
FUNCTION_BLOCK "A_3125_MXZ01MA_Code"
TITLE =A_3125_MXZ01MA FAN 1
//COPYRIGHT:     (C) 2009  BUHLER AG, CH-9240 UZWIL, SWITZERLAND
//
//PRODUCT:       WinCoS_BIW01_09
//
//TITLE:         FAN 1
//
//--------------------------------------------------------------------------------
//
//IDENT:         AUTHOR:             DEPT:                             DATE:
//
//P01_FB1018.1.0 K.Renz              CSB41                             20.Mai.2010
//               1st Release
//
//--------------------------------------------------------------------------------
//
//PURPOSE:
//
//MANUAL :
//
//RESTRICTIONS:
//
//--------------------------------------------------------------------------------
AUTHOR : KR
FAMILY : USW
VERSION : 0.0


VAR
  Ma : "GCS7_M_FB50_Data";	// Machine
  A_3125_KCU04 : "GCS7_E_DigInput";	// Mon1: DigInpCont
  Mon2 : "GCS7_E_DigInput";	// Mon2: DigInpCont
  Mon3 : "GCS7_E_DigInput";	// spare
  A_3125_BSA07 : "GCS7_E_DigInput";	// Mon4: DigInpCont
  Mon5 : "GCS7_E_DigInput";	// spare
  Mon6 : "GCS7_E_DigInput";	// spare
  A_3125_MXZ01 : "GCS7_E_Motor";	// Motor: Motor
END_VAR
BEGIN
NETWORK
TITLE =Call SSW

      UC    "GCS7_M_Motor6Mon";
END_FUNCTION_BLOCK


FUNCTION_BLOCK "A_3126_MXZ01MA_Code"
TITLE =A_3126_MXZ01MA FAN 2
//COPYRIGHT:     (C) 2009  BUHLER AG, CH-9240 UZWIL, SWITZERLAND
//
//PRODUCT:       WinCoS_BIW01_09
//
//TITLE:         FAN 2
//
//--------------------------------------------------------------------------------
//
//IDENT:         AUTHOR:             DEPT:                             DATE:
//
//P01_FB1019.1.0 K.Renz              CSB41                             20.Mai.2010
//               1st Release
//
//--------------------------------------------------------------------------------
//
//PURPOSE:
//
//MANUAL :
//
//RESTRICTIONS:
//
//--------------------------------------------------------------------------------
AUTHOR : KR
FAMILY : USW
VERSION : 0.0


VAR
  Ma : "GCS7_M_FB50_Data";	// Machine
  A_3126_KCU04 : "GCS7_E_DigInput";	// Mon1: DigInpCont
  Mon2 : "GCS7_E_DigInput";	// Mon2: DigInpCont
  Mon3 : "GCS7_E_DigInput";	// spare
  A_3126_BSA07 : "GCS7_E_DigInput";	// Mon4: DigInpCont
  Mon5 : "GCS7_E_DigInput";	// spare
  Mon6 : "GCS7_E_DigInput";	// spare
  A_3126_MXZ01 : "GCS7_E_Motor";	// Motor: Motor
END_VAR
BEGIN
NETWORK
TITLE =Call SSW

      UC    "GCS7_M_Motor6Mon";
END_FUNCTION_BLOCK


FUNCTION_BLOCK "A_3914_MXZ01MA_Code"
TITLE =A_3125_MXZ02MA GETRIEBEÖLPUMPE FAN 1
//COPYRIGHT:     (C) 2009  BUHLER AG, CH-9240 UZWIL, SWITZERLAND
//
//PRODUCT:       WinCoS_BIW01_09
//
//TITLE:         GETRIEBEÖLPUMPE FAN 1
//
//--------------------------------------------------------------------------------
//
//IDENT:         AUTHOR:             DEPT:                             DATE:
//
//P01_FB1025.1.0 K.Renz              CSB41                             20.Mai.2010
//               1st Release
//
//--------------------------------------------------------------------------------
//
//PURPOSE:
//
//MANUAL :
//
//RESTRICTIONS:
//
//--------------------------------------------------------------------------------
AUTHOR : KR
FAMILY : USW
VERSION : 0.0


VAR
  Ma : "GCS7_M_FB50_Data";	// Machine
  A_3125_BFT09 : "GCS7_E_DigInput";	// Mon1: DigInpCont
  Mon2 : "GCS7_E_DigInput";	// Mon2: DigInpCont
  Mon3 : "GCS7_E_DigInput";	// spare
  Mon4 : "GCS7_E_DigInput";	// spare
  Mon5 : "GCS7_E_DigInput";	// spare
  Mon6 : "GCS7_E_DigInput";	// spare
  A_3125_MXZ02 : "GCS7_E_Motor";	// Motor: Motor
END_VAR
BEGIN
NETWORK
TITLE =Call SSW

      UC    "GCS7_M_Motor6Mon";
END_FUNCTION_BLOCK


FUNCTION_BLOCK FB 1065
TITLE =A_3126_MXZ02MA GETRIEBEÖLPUMPE FAN 2
//COPYRIGHT:     (C) 2009  BUHLER AG, CH-9240 UZWIL, SWITZERLAND
//
//PRODUCT:       WinCoS_BIW01_09
//
//TITLE:         GETRIEBEÖLPUMPE FAN 2
//
//--------------------------------------------------------------------------------
//
//IDENT:         AUTHOR:             DEPT:                             DATE:
//
//P01_FB1065.1.0 K.Renz              CSB41                             20.Mai.2010
//               1st Release
//
//--------------------------------------------------------------------------------
//
//PURPOSE:
//
//MANUAL :
//
//RESTRICTIONS:
//
//--------------------------------------------------------------------------------
AUTHOR : KR
FAMILY : USW
VERSION : 0.0


VAR
  Ma : "GCS7_M_FB50_Data";	// Machine
  A_3225_BFT09 : "GCS7_E_DigInput";	// Mon1: DigInpCont
  Mon2 : "GCS7_E_DigInput";	// Mon2: DigInpCont
  Mon3 : "GCS7_E_DigInput";	// spare
  Mon4 : "GCS7_E_DigInput";	// spare
  Mon5 : "GCS7_E_DigInput";	// spare
  Mon6 : "GCS7_E_DigInput";	// spare
  A_3225_MXZ02 : "GCS7_E_Motor";	// Motor: Motor
END_VAR
BEGIN
NETWORK
TITLE =Call SSW

      UC    "GCS7_M_Motor6Mon";
END_FUNCTION_BLOCK


FUNCTION_BLOCK "G271M_Code"
TITLE =G271M FAN KILN 1
//COPYRIGHT:    (C) 2009  BUHLER AG, CH-9240 UZWIL, SWITZERLAND
//
//PRODUCT:      WinCoS_BIW01_09
//
//TITLE:        FAN KILN 1
//                Machine group control
//                Maschinengruppensteuerung
//
//--------------------------------------------------------------------------------
//
//IDENT:        AUTHOR:             DEPT:                              DATE:
//
//P01_FB371.1.0 K.Renz              CSB41                              20.Mai.2010
//             1st Release
//
//--------------------------------------------------------------------------------
//
//PURPOSE:
//
//MANUAL :
//
//RESTRICTIONS:
//
//--------------------------------------------------------------------------------
AUTHOR : KR
FAMILY : USW
VERSION : 9.9


VAR
  Gr : "GCS7_GrpCtrlSub";	//Standard interface to group
  InOutValue1 : DINT ;	//Data for user
  InOutValue2 : DINT ;	//Data for user
  OutWayConflict : BOOL ;	//Data for user
  OutSelectionOk : BOOL ;	//Data for user
  CmdNewValue : BOOL ;	//Data for user
  CmdNewJob : BOOL ;	//Data for user
  OutCodeOK : BOOL ;	//Data for user
  InEndOfJob : BOOL ;	//Data for user
  staWayOk : BOOL ;	//Data for user
  EdgeStartRelease : BOOL ;	//Data for user
  USW8 : BOOL ;	//Data for user
  USW9 : BOOL ;	//Data for user
  USW10 : BOOL ;	//Data for user
  USW11 : BOOL ;	//Data for user
  USW12 : BOOL ;	//Data for user
  USW13 : BOOL ;	//Data for user
  USW14 : BOOL ;	//Data for user
  USW15 : BOOL ;	//Data for user
  A_3125_KCU04AI1 : "GCS7_E_AnalogInput";	// AnaInp
  A_3125_KCU04AI2 : "GCS7_E_AnalogInput";	// AnaInp
  A_3125_BTE05 : "GCS7_E_AnalogInput";	// AnaInp
  A_3125_BTE06 : "GCS7_E_AnalogInput";	// AnaInp
  A_3125_MXZ01MA : "A_3125_MXZ01MA_Code";	// Motor+6DI
  A_3125_TSC01_COM : "SSA_ABB";	// FU_ABB
  A_3125_TSC01_AC : "GCS7_E_AnalogInput";	// AnaInp
  A_3125_TSC01_AF : "GCS7_E_AnalogInput";	// AnaInp
  A_3125_TSC01_AT : "GCS7_E_AnalogInput";	// AnaInp
  A_3125_TSC01_AP : "GCS7_E_AnalogInput";	// AnaInp
  A_3126_KCU04AI1 : "GCS7_E_AnalogInput";	// AnaInp
  A_3126_KCU04AI2 : "GCS7_E_AnalogInput";	// AnaInp
  A_3126_BTE05 : "GCS7_E_AnalogInput";	// AnaInp
  A_3126_BTE06 : "GCS7_E_AnalogInput";	// AnaInp
  A_3126_MXZ01MA : "A_3126_MXZ01MA_Code";	// Motor+6DI
  A_3126_TSC01_COM : "SSA_ABB";	// FU_ABB
  A_3126_TSC01_AC : "GCS7_E_AnalogInput";	// AnaInp
  A_3126_TSC01_AF : "GCS7_E_AnalogInput";	// AnaInp
  A_3126_TSC01_AP : "GCS7_E_AnalogInput";	// AnaInp
  A_3126_TSC01_AT : "GCS7_E_AnalogInput";	// AnaInp
  A_3125_TSC01 : "GCS7_E_DigInput";	// DigInpCont
  A_3126_TSC01 : "GCS7_E_DigInput";	// DigInpCont
  A_3125_MXZ02MA : "A_3914_MXZ01MA_Code";	// Motor+6DI
  A_3126_MXZ02MA : FB 1065;	// Motor+6DI
END_VAR
VAR_TEMP
  tmpEnable : BOOL ;
  tmpFlag : BOOL ;
  tmpCmdNext : BOOL ;
  tmpLocal : BOOL ;
  tmpAspOk : BOOL ;
  tmpHWStop : BOOL ;
  tmpInstanzDBNo : INT ;
END_VAR
BEGIN
NETWORK
TITLE =

NETWORK
TITLE =Read command from group control
//Parameter
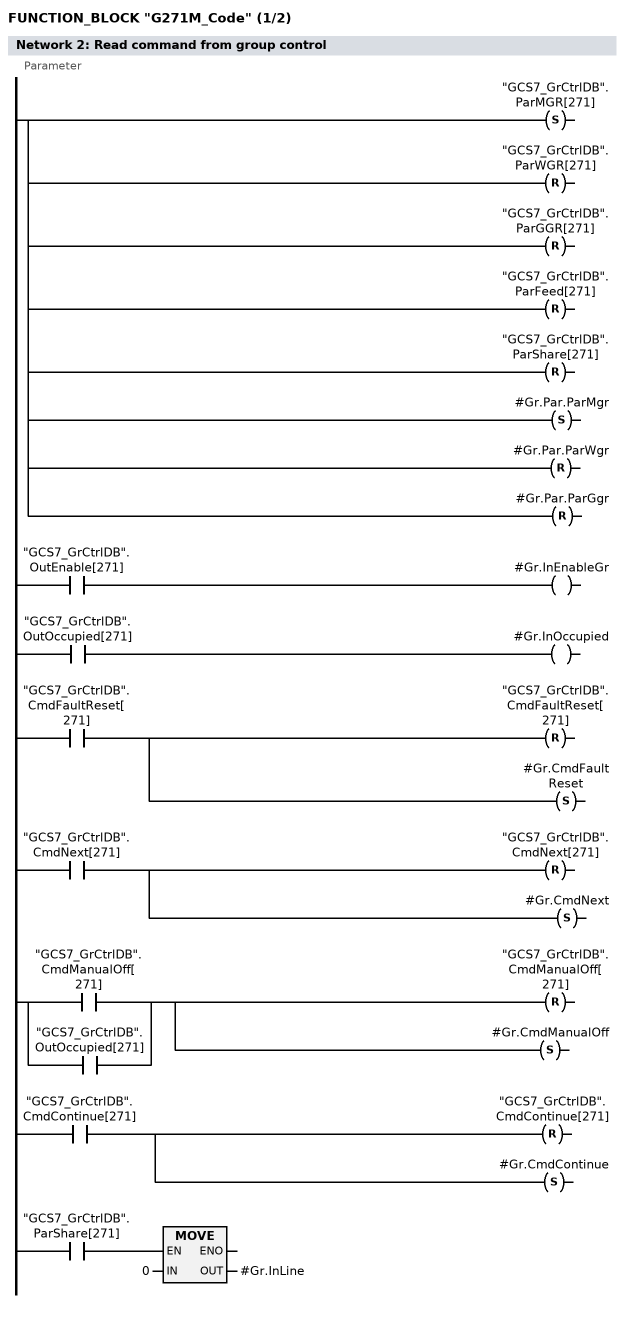
      SET   ;
      S     "GCS7_GrCtrlDB".ParMGR[271];
      R     "GCS7_GrCtrlDB".ParWGR[271];
      R     "GCS7_GrCtrlDB".ParGGR[271];
      R     "GCS7_GrCtrlDB".ParFeed[271];
      R     "GCS7_GrCtrlDB".ParShare[271];
      S     #Gr.Par.ParMgr;
      R     #Gr.Par.ParWgr;
      R     #Gr.Par.ParGgr;
//Command
      U     "GCS7_GrCtrlDB".OutEnable[271];
      =     #Gr.InEnableGr;
      U     "GCS7_GrCtrlDB".OutOccupied[271];
      =     #Gr.InOccupied;
      U     "GCS7_GrCtrlDB".CmdFaultReset[271];
      R     "GCS7_GrCtrlDB".CmdFaultReset[271];
      S     #Gr.CmdFaultReset;
      U     "GCS7_GrCtrlDB".CmdNext[271];
      R     "GCS7_GrCtrlDB".CmdNext[271];
      S     #Gr.CmdNext;
      U     "GCS7_GrCtrlDB".CmdManualOff[271];
      O     "GCS7_GrCtrlDB".OutOccupied[271];
      R     "GCS7_GrCtrlDB".CmdManualOff[271];
      S     #Gr.CmdManualOff;
      U     "GCS7_GrCtrlDB".CmdContinue[271];
      R     "GCS7_GrCtrlDB".CmdContinue[271];
      S     #Gr.CmdContinue;
//Init Line Number
      U     "GCS7_GrCtrlDB".ParShare[271];
      SPBN  WE00;
      L     0;
      T     #Gr.InLine;
WE00: NOP   0;
NETWORK
TITLE =Call Methode Control
// 1. Handle Interface PCControl
// 2. Prepare mode --> ModePassive,ModeActive,ModeIdling
// 3. Reset global flags of the group
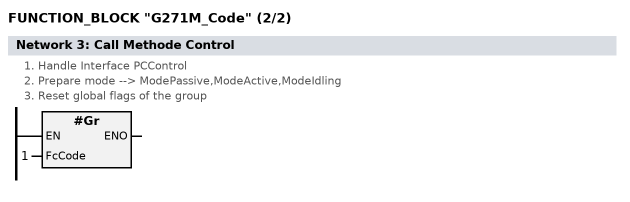
      CALL #Gr (
           FcCode                   := 1);
NETWORK
TITLE =Restart Idling Time

      L     #Gr.Par.ParIdling;
      L     2;
      >=I   ;
      SPB   IdTm;
      T     #Gr.Par.ParIdling;
IdTm: NOP   0;
      CLR   ;
      S     #Gr.CmdRestartIdling;
NETWORK
TITLE =Prepare global flags

NETWORK
TITLE =Set Pattern (Target position)

NETWORK
TITLE =Interlocking WayOk

NETWORK
TITLE =Interlocking Autostart

      CLR   ;
      R     #Gr.OutAutostart;
NETWORK
TITLE =Interlocking Enable
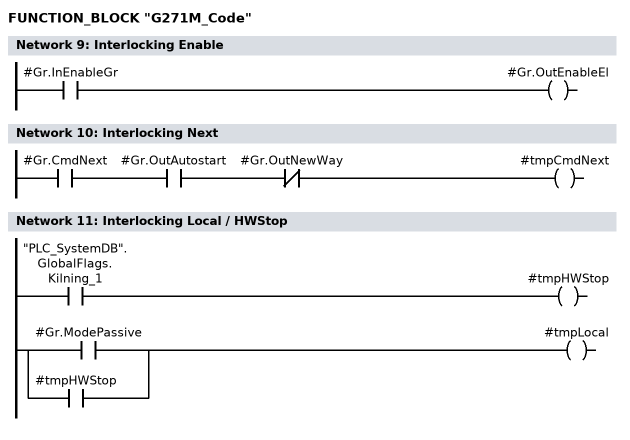

      U     #Gr.InEnableGr;
      =     #Gr.OutEnableEl;

NETWORK
TITLE =Interlocking Next

      U     #Gr.CmdNext;
      U     #Gr.OutAutostart;
      UN    #Gr.OutNewWay;
      =     #tmpCmdNext;

NETWORK
TITLE =Interlocking Local / HWStop

      U     "PLC_SystemDB".GlobalFlags.Kilning_1;
      =     #tmpHWStop;

      U     #Gr.ModePassive;
      O     #tmpHWStop;
      =     #tmpLocal;

NETWORK
TITLE =Interlocking Start Warning

      NOP   0;
//- Restart after fault --
      U     #Gr.CmdFaultReset;
      U     #Gr.VarFault;
      S     "SYS_StartWarningDB".Area[10].CmdResetStartWarning;
//- Run Timer --
      AUF   "G271M";
      CALL "GCS7_StartWarning" , "SYS_StartWarningDB" (
           InModeHigher             := FALSE,
           InArea                   := 10,
           InEnable                 := #Gr.OutEnableEl,
           InLocal                  := #tmpLocal,
           InStarted                := #Gr.VarStarted,
           InCmdNext                := #tmpCmdNext,
           OutCmdNext               := #tmpCmdNext,
           OutStartwarning          := #Gr.VarStartwarning);
//- Store Startwarning done  --
//- Reset Autostart --
      U     "SYS_StartWarningDB".TmpArea.OutStartReleaseRunningL;
      FN    #EdgeStartRelease;
      U     #Gr.VarFault;
      R     #Gr.OutAutostart;
NETWORK
TITLE ==A-3125-KCU04AI1 : VIBRATION MONITOR FAN 1 CHANNEL 1

      NOP   0;
//-InLocal---
      U     #tmpLocal;
      =     #A_3125_KCU04AI1.InLocal;
//
//-Monitoring---
      CLR   ;
      =     #A_3125_KCU04AI1.InMonLL;
      CLR   ;
      =     #A_3125_KCU04AI1.InMonL;
      CLR   ;
      =     #A_3125_KCU04AI1.InMonMid;
      CLR   ;
      =     #A_3125_KCU04AI1.InMonH;
      SET   ;
      =     #A_3125_KCU04AI1.InMonHH;
//
//-Read inputs---
      L     "A_3125_KCU04_AI1";
      T     #A_3125_KCU04AI1.InpValue;
      U     "PLC_SystemDB".GlobalFlags.Kilning_1;
      =     #A_3125_KCU04AI1.InHWStop;
      U     "PLC_DPInfo".Master[1].SlavesError[92];
      =     #A_3125_KCU04AI1.InDPFault;
//
//-Set Parameters---
//
//-Call object control---
      CALL #A_3125_KCU04AI1 ;
//
//-Write outputs---
NETWORK
TITLE ==A-3125-KCU04AI2 : VIBRATION MONITOR FAN 1 CHANNEL 2

      NOP   0;
//-InLocal---
      U     #tmpLocal;
      =     #A_3125_KCU04AI2.InLocal;
//
//-Monitoring---
      CLR   ;
      =     #A_3125_KCU04AI2.InMonLL;
      CLR   ;
      =     #A_3125_KCU04AI2.InMonL;
      CLR   ;
      =     #A_3125_KCU04AI2.InMonMid;
      CLR   ;
      =     #A_3125_KCU04AI2.InMonH;
      SET   ;
      =     #A_3125_KCU04AI2.InMonHH;
//
//-Read inputs---
      L     "A_3125_KCU04_AI2";
      T     #A_3125_KCU04AI2.InpValue;
      U     "PLC_SystemDB".GlobalFlags.Kilning_1;
      =     #A_3125_KCU04AI2.InHWStop;
      U     "PLC_DPInfo".Master[1].SlavesError[92];
      =     #A_3125_KCU04AI2.InDPFault;
//
//-Set Parameters---
//
//-Call object control---
      CALL #A_3125_KCU04AI2 ;
//
//-Write outputs---
NETWORK
TITLE ==A-3125-BTE05 : TEMPERATURE BEARING TEMPERATUR SENSOR

      NOP   0;
//-InLocal---
      U     #tmpLocal;
      =     #A_3125_BTE05.InLocal;
//
//-Monitoring---
      CLR   ;
      =     #A_3125_BTE05.InMonLL;
      CLR   ;
      =     #A_3125_BTE05.InMonL;
      CLR   ;
      =     #A_3125_BTE05.InMonMid;
      CLR   ;
      =     #A_3125_BTE05.InMonH;
      SET   ;
      =     #A_3125_BTE05.InMonHH;
//
//-Read inputs---
      L     "A_3125_BTE05_AI1";
      T     #A_3125_BTE05.InpValue;
      U     "PLC_SystemDB".GlobalFlags.Kilning_1;
      =     #A_3125_BTE05.InHWStop;
      U     "PLC_DPInfo".Master[1].SlavesError[92];
      =     #A_3125_BTE05.InDPFault;
//
//-Set Parameters---
//
//-Call object control---
      CALL #A_3125_BTE05 ;
//
//-Write outputs---
NETWORK
TITLE ==A-3125-BTE06 : TEMPERATURE BEARING TEMPERATUR SENSOR

      NOP   0;
//-InLocal---
      U     #tmpLocal;
      =     #A_3125_BTE06.InLocal;
//
//-Monitoring---
      CLR   ;
      =     #A_3125_BTE06.InMonLL;
      CLR   ;
      =     #A_3125_BTE06.InMonL;
      CLR   ;
      =     #A_3125_BTE06.InMonMid;
      CLR   ;
      =     #A_3125_BTE06.InMonH;
      SET   ;
      =     #A_3125_BTE06.InMonHH;
//
//-Read inputs---
      L     "A_3125_BTE06_AI1";
      T     #A_3125_BTE06.InpValue;
      U     "PLC_SystemDB".GlobalFlags.Kilning_1;
      =     #A_3125_BTE06.InHWStop;
      U     "PLC_DPInfo".Master[1].SlavesError[92];
      =     #A_3125_BTE06.InDPFault;
//
//-Set Parameters---
//
//-Call object control---
      CALL #A_3125_BTE06 ;
//
//-Write outputs---
NETWORK
TITLE ==A-3125-MXZ02MA : GETRIEBEÖLPUMPE FAN 1
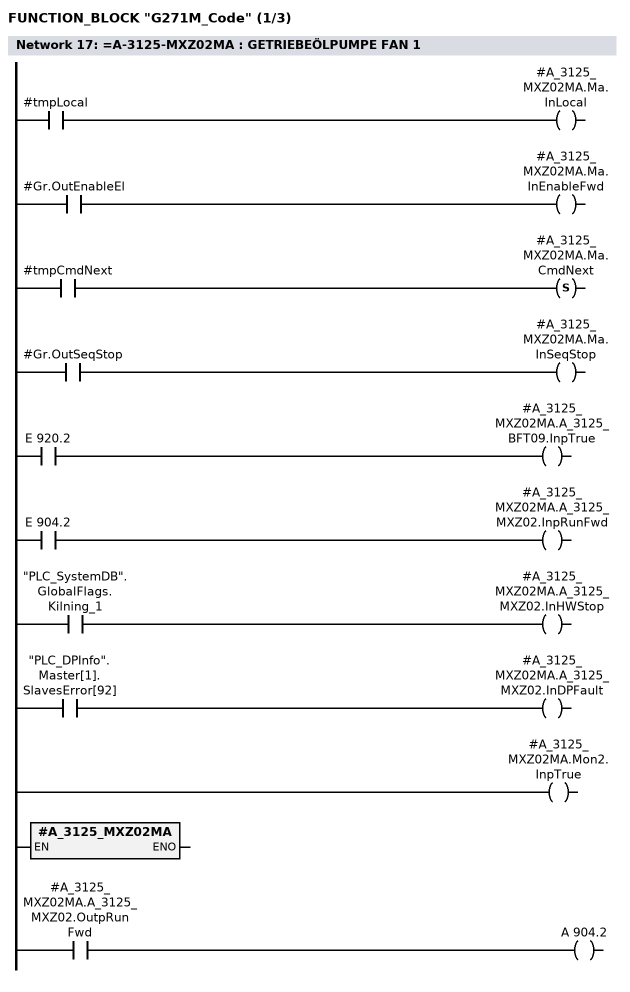

      NOP   0;
//-InLocal---
      U     #tmpLocal;
      =     #A_3125_MXZ02MA.Ma.InLocal;
//
//-Interlocking---

      U     #Gr.OutEnableEl;
      =     #A_3125_MXZ02MA.Ma.InEnableFwd;
//
      U     #tmpCmdNext;
      S     #A_3125_MXZ02MA.Ma.CmdNext;
//
      U     #Gr.OutSeqStop;
      =     #A_3125_MXZ02MA.Ma.InSeqStop;
//
//=Values and commands of elements===
//-=A-3125-BFT09---
//      CLR
//      S     #A_3125_MXZ02MA.A_3125_BFT09.CmdRunTimeOutTime
//
//-Read inputs of elements---
      U     E    920.2;
      =     #A_3125_MXZ02MA.A_3125_BFT09.InpTrue;
      U     E    904.2;
      =     #A_3125_MXZ02MA.A_3125_MXZ02.InpRunFwd;
      U     "PLC_SystemDB".GlobalFlags.Kilning_1;
      =     #A_3125_MXZ02MA.A_3125_MXZ02.InHWStop;
      U     "PLC_DPInfo".Master[1].SlavesError[92];
      =     #A_3125_MXZ02MA.A_3125_MXZ02.InDPFault;
      SET   ;
      =     #A_3125_MXZ02MA.Mon2.InpTrue;
//
//-Set Parameters---
//
//-Call object control---
      CALL #A_3125_MXZ02MA ;
//
//-Write outputs---
      U     #A_3125_MXZ02MA.A_3125_MXZ02.OutpRunFwd;
      =     A    904.2;
NETWORK
TITLE ==A-3125-MXZ01MA : FAN 1
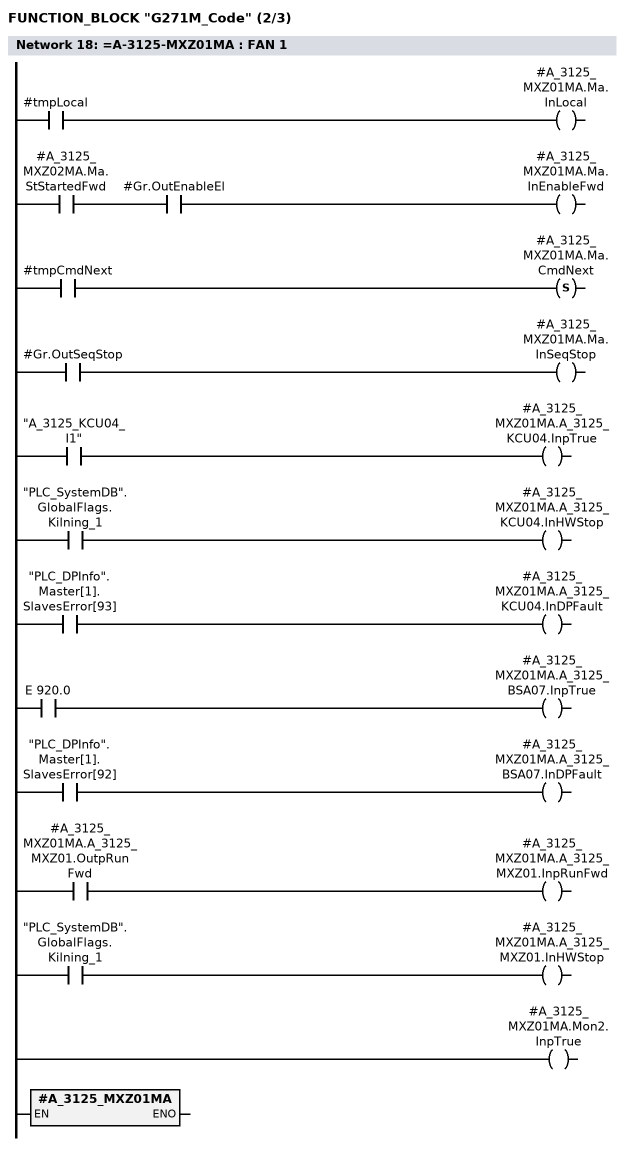

      NOP   0;
//-InLocal---
      U     #tmpLocal;
      =     #A_3125_MXZ01MA.Ma.InLocal;
//
//-Interlocking---
      U     #A_3125_MXZ02MA.Ma.StStartedFwd;
      U     #Gr.OutEnableEl;
      =     #A_3125_MXZ01MA.Ma.InEnableFwd;
//
      U     #tmpCmdNext;
      S     #A_3125_MXZ01MA.Ma.CmdNext;
//
      U     #Gr.OutSeqStop;
      =     #A_3125_MXZ01MA.Ma.InSeqStop;
//
//=Values and commands of elements===
//-=A-3125-KCU04---
//      CLR
//      S     #A_3125_MXZ01MA.A_3125_KCU04.CmdRunTimeOutTime
//-=A-3125-BSA07---
//      CLR
//      S     #A_3125_MXZ01MA.A_3125_BSA07.CmdRunTimeOutTime
//
//-Read inputs of elements---
      U     "A_3125_KCU04_I1";
      =     #A_3125_MXZ01MA.A_3125_KCU04.InpTrue;
      U     "PLC_SystemDB".GlobalFlags.Kilning_1;
      =     #A_3125_MXZ01MA.A_3125_KCU04.InHWStop;
      U     "PLC_DPInfo".Master[1].SlavesError[93];
      =     #A_3125_MXZ01MA.A_3125_KCU04.InDPFault;
      U     E    920.0;
      =     #A_3125_MXZ01MA.A_3125_BSA07.InpTrue;
      U     "PLC_DPInfo".Master[1].SlavesError[92];
      =     #A_3125_MXZ01MA.A_3125_BSA07.InDPFault;
      U     #A_3125_MXZ01MA.A_3125_MXZ01.OutpRunFwd;
      =     #A_3125_MXZ01MA.A_3125_MXZ01.InpRunFwd;
      U     "PLC_SystemDB".GlobalFlags.Kilning_1;
      =     #A_3125_MXZ01MA.A_3125_MXZ01.InHWStop;
      SET   ;
      =     #A_3125_MXZ01MA.Mon2.InpTrue;
//
//-Set Parameters---
//
//-Call object control---
      CALL #A_3125_MXZ01MA ;
//
//-Write outputs---
NETWORK
TITLE ==A-3125-TSC01_COM : FAN 1 FU KOMMUNIKATION
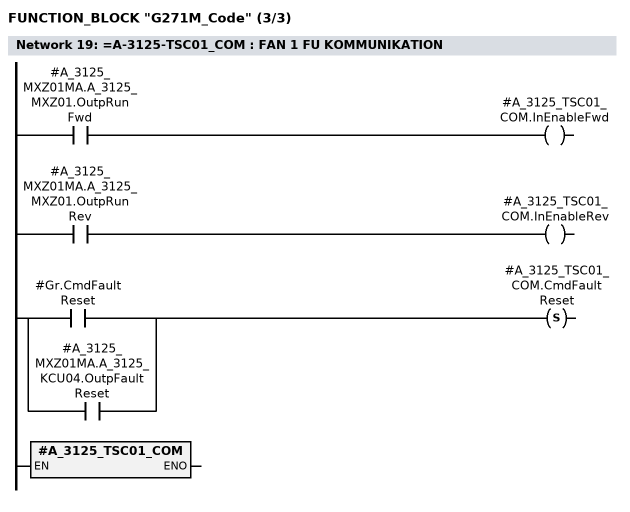

      NOP   0;
      U     #A_3125_MXZ01MA.A_3125_MXZ01.OutpRunFwd;
      =     #A_3125_TSC01_COM.InEnableFwd;
      U     #A_3125_MXZ01MA.A_3125_MXZ01.OutpRunRev;
      =     #A_3125_TSC01_COM.InEnableRev;
      U     #Gr.CmdFaultReset;
      O     #A_3125_MXZ01MA.A_3125_KCU04.OutpFaultReset;
      S     #A_3125_TSC01_COM.CmdFaultReset;
//
//
//-Read inputs---
//
//-Set Parameters---
//
//-Call object control---
      CALL #A_3125_TSC01_COM ;
//
//-Write outputs---
NETWORK
TITLE ==A-3125-TSC01_AC : ACT. CURRENT FAN 1 FU

      NOP   0;
//-InLocal---
      U     #tmpLocal;
      =     #A_3125_TSC01_AC.InLocal;
//
//-Monitoring---
      SET   ;
      =     #A_3125_TSC01_AC.InMonLL;
      CLR   ;
      =     #A_3125_TSC01_AC.InMonL;
      CLR   ;
      =     #A_3125_TSC01_AC.InMonMid;
      CLR   ;
      =     #A_3125_TSC01_AC.InMonH;
      CLR   ;
      =     #A_3125_TSC01_AC.InMonHH;
//
//-Read inputs---
      L     #A_3125_TSC01_COM.Output.SetpointValue01;
      ITD   ;
      DTR   ;
      ABS   ;
      RND   ;
      T     #A_3125_TSC01_AC.InpValue;
      U     "PLC_SystemDB".GlobalFlags.Kilning_1;
      =     #A_3125_TSC01_AC.InHWStop;
//
//-Set Parameters---
//
//-Call object control---
      CALL #A_3125_TSC01_AC ;
//
//-Write outputs---
NETWORK
TITLE ==A-3125-TSC01_AF : ACT. FREQUENCY FAN 1 FU

      NOP   0;
//-InLocal---
      U     #tmpLocal;
      =     #A_3125_TSC01_AF.InLocal;
//
//-Monitoring---
      SET   ;
      =     #A_3125_TSC01_AF.InMonLL;
      CLR   ;
      =     #A_3125_TSC01_AF.InMonL;
      CLR   ;
      =     #A_3125_TSC01_AF.InMonMid;
      CLR   ;
      =     #A_3125_TSC01_AF.InMonH;
      CLR   ;
      =     #A_3125_TSC01_AF.InMonHH;
//
//-Read inputs---
      L     #A_3125_TSC01_COM.Output.SetpointValue01;
      ITD   ;
      DTR   ;
      ABS   ;
      RND   ;
      T     #A_3125_TSC01_AF.InpValue;
      U     "PLC_SystemDB".GlobalFlags.Kilning_1;
      =     #A_3125_TSC01_AF.InHWStop;
//
//-Set Parameters---
//
//-Call object control---
      CALL #A_3125_TSC01_AF ;
//
//-Write outputs---
NETWORK
TITLE ==A-3125-TSC01_AT : ACT. TORQUE FAN 1 FU

      NOP   0;
//-InLocal---
      U     #tmpLocal;
      =     #A_3125_TSC01_AT.InLocal;
//
//-Monitoring---
      CLR   ;
      =     #A_3125_TSC01_AT.InMonLL;
      CLR   ;
      =     #A_3125_TSC01_AT.InMonL;
      CLR   ;
      =     #A_3125_TSC01_AT.InMonMid;
      CLR   ;
      =     #A_3125_TSC01_AT.InMonH;
      CLR   ;
      =     #A_3125_TSC01_AT.InMonHH;
//
//-Read inputs---
      L     #A_3125_TSC01_COM.Output.SetpointValue01;
      ITD   ;
      DTR   ;
      ABS   ;
      RND   ;
      T     #A_3125_TSC01_AT.InpValue;
      U     "PLC_SystemDB".GlobalFlags.Kilning_1;
      =     #A_3125_TSC01_AT.InHWStop;
//
//-Set Parameters---
//
//-Call object control---
      CALL #A_3125_TSC01_AT ;
//
//-Write outputs---
NETWORK
TITLE ==A-3125-TSC01_AP : ACT. POWER FAN 1 FU

      NOP   0;
//-InLocal---
      U     #tmpLocal;
      =     #A_3125_TSC01_AP.InLocal;
//
//-Monitoring---
      CLR   ;
      =     #A_3125_TSC01_AP.InMonLL;
      CLR   ;
      =     #A_3125_TSC01_AP.InMonL;
      CLR   ;
      =     #A_3125_TSC01_AP.InMonMid;
      CLR   ;
      =     #A_3125_TSC01_AP.InMonH;
      CLR   ;
      =     #A_3125_TSC01_AP.InMonHH;
//
//-Read inputs---
      L     #A_3125_TSC01_COM.Output.SetpointValue01;
      ITD   ;
      DTR   ;
      ABS   ;
      RND   ;
      T     #A_3125_TSC01_AP.InpValue;
      U     "PLC_SystemDB".GlobalFlags.Kilning_1;
      =     #A_3125_TSC01_AP.InHWStop;
//
//-Set Parameters---
//
//-Call object control---
      CALL #A_3125_TSC01_AP ;
//
//-Write outputs---
NETWORK
TITLE ==A-3126-KCU04AI1 : VIBRATION MONITOR FAN 2 CHANNEL 1

      NOP   0;
//-InLocal---
      U     #tmpLocal;
      =     #A_3126_KCU04AI1.InLocal;
//
//-Monitoring---
      CLR   ;
      =     #A_3126_KCU04AI1.InMonLL;
      CLR   ;
      =     #A_3126_KCU04AI1.InMonL;
      CLR   ;
      =     #A_3126_KCU04AI1.InMonMid;
      CLR   ;
      =     #A_3126_KCU04AI1.InMonH;
      SET   ;
      =     #A_3126_KCU04AI1.InMonHH;
//
//-Read inputs---
      L     "A_3126_KCU04_AI1";
      T     #A_3126_KCU04AI1.InpValue;
      U     "PLC_SystemDB".GlobalFlags.Kilning_1;
      =     #A_3126_KCU04AI1.InHWStop;
      U     "PLC_DPInfo".Master[1].SlavesError[92];
      =     #A_3126_KCU04AI1.InDPFault;
//
//-Set Parameters---
//
//-Call object control---
      CALL #A_3126_KCU04AI1 ;
//
//-Write outputs---
NETWORK
TITLE ==A-3126-KCU04AI2 : VIBRATION MONITOR FAN 2 CHANNEL 2

      NOP   0;
//-InLocal---
      U     #tmpLocal;
      =     #A_3126_KCU04AI2.InLocal;
//
//-Monitoring---
      CLR   ;
      =     #A_3126_KCU04AI2.InMonLL;
      CLR   ;
      =     #A_3126_KCU04AI2.InMonL;
      CLR   ;
      =     #A_3126_KCU04AI2.InMonMid;
      CLR   ;
      =     #A_3126_KCU04AI2.InMonH;
      SET   ;
      =     #A_3126_KCU04AI2.InMonHH;
//
//-Read inputs---
      L     "A_3126_KCU04_AI2";
      T     #A_3126_KCU04AI2.InpValue;
      U     "PLC_SystemDB".GlobalFlags.Kilning_1;
      =     #A_3126_KCU04AI2.InHWStop;
      U     "PLC_DPInfo".Master[1].SlavesError[92];
      =     #A_3126_KCU04AI2.InDPFault;
//
//-Set Parameters---
//
//-Call object control---
      CALL #A_3126_KCU04AI2 ;
//
//-Write outputs---
NETWORK
TITLE ==A-3126-BTE05 : TEMPERATURE BEARING TEMPERATUR SENSOR

      NOP   0;
//-InLocal---
      U     #tmpLocal;
      =     #A_3126_BTE05.InLocal;
//
//-Monitoring---
      CLR   ;
      =     #A_3126_BTE05.InMonLL;
      CLR   ;
      =     #A_3126_BTE05.InMonL;
      CLR   ;
      =     #A_3126_BTE05.InMonMid;
      CLR   ;
      =     #A_3126_BTE05.InMonH;
      SET   ;
      =     #A_3126_BTE05.InMonHH;
//
//-Read inputs---
      L     "A_3126_BTE05_AI1";
      T     #A_3126_BTE05.InpValue;
      U     "PLC_SystemDB".GlobalFlags.Kilning_1;
      =     #A_3126_BTE05.InHWStop;
      U     "PLC_DPInfo".Master[1].SlavesError[92];
      =     #A_3126_BTE05.InDPFault;
//
//-Set Parameters---
//
//-Call object control---
      CALL #A_3126_BTE05 ;
//
//-Write outputs---
NETWORK
TITLE ==A-3126-BTE06 : TEMPERATURE BEARING TEMPERATUR SENSOR

      NOP   0;
//-InLocal---
      U     #tmpLocal;
      =     #A_3126_BTE06.InLocal;
//
//-Monitoring---
      CLR   ;
      =     #A_3126_BTE06.InMonLL;
      CLR   ;
      =     #A_3126_BTE06.InMonL;
      CLR   ;
      =     #A_3126_BTE06.InMonMid;
      CLR   ;
      =     #A_3126_BTE06.InMonH;
      SET   ;
      =     #A_3126_BTE06.InMonHH;
//
//-Read inputs---
      L     "A_3126_BTE06_AI1";
      T     #A_3126_BTE06.InpValue;
      U     "PLC_SystemDB".GlobalFlags.Kilning_1;
      =     #A_3126_BTE06.InHWStop;
      U     "PLC_DPInfo".Master[1].SlavesError[92];
      =     #A_3126_BTE06.InDPFault;
//
//-Set Parameters---
//
//-Call object control---
      CALL #A_3126_BTE06 ;
//
//-Write outputs---
NETWORK
TITLE ==A-3126-MXZ02MA : GETRIEBEÖLPUMPE FAN 2
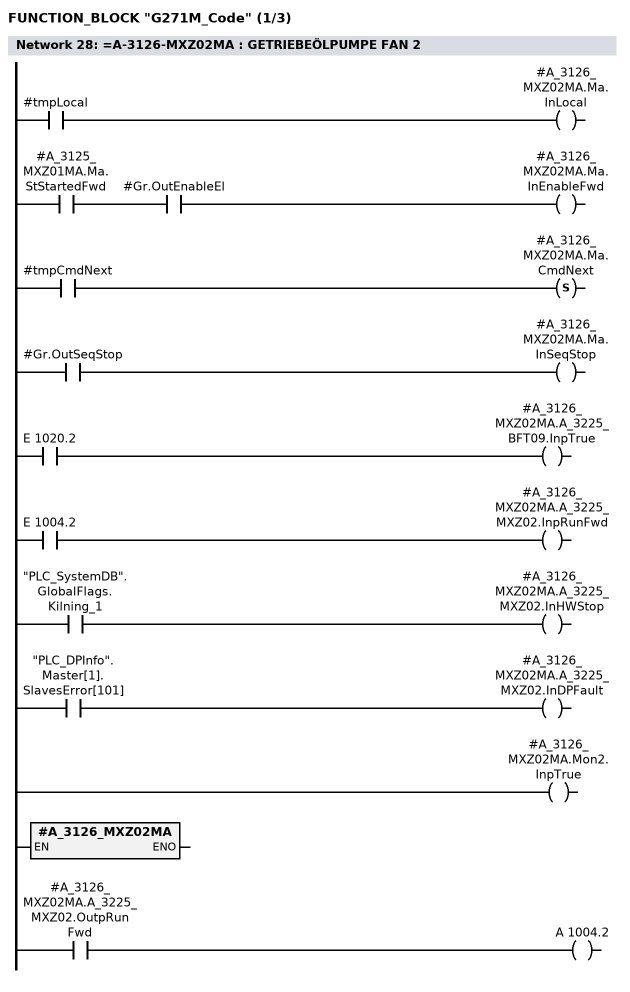

      NOP   0;
//-InLocal---
      U     #tmpLocal;
      =     #A_3126_MXZ02MA.Ma.InLocal;
//
//-Interlocking---
      U     #A_3125_MXZ01MA.Ma.StStartedFwd;
      U     #Gr.OutEnableEl;
      =     #A_3126_MXZ02MA.Ma.InEnableFwd;
//
      U     #tmpCmdNext;
      S     #A_3126_MXZ02MA.Ma.CmdNext;
//
      U     #Gr.OutSeqStop;
      =     #A_3126_MXZ02MA.Ma.InSeqStop;
//
//=Values and commands of elements===
//-=A-3225-BFT09---
//      CLR
//      S     #A_3126_MXZ02MA.A_3225_BFT09.CmdRunTimeOutTime
//
//-Read inputs of elements---
      U     E   1020.2;
      =     #A_3126_MXZ02MA.A_3225_BFT09.InpTrue;
      U     E   1004.2;
      =     #A_3126_MXZ02MA.A_3225_MXZ02.InpRunFwd;
      U     "PLC_SystemDB".GlobalFlags.Kilning_1;
      =     #A_3126_MXZ02MA.A_3225_MXZ02.InHWStop;
      U     "PLC_DPInfo".Master[1].SlavesError[101];
      =     #A_3126_MXZ02MA.A_3225_MXZ02.InDPFault;
      SET   ;
      =     #A_3126_MXZ02MA.Mon2.InpTrue;
//
//-Set Parameters---
//
//-Call object control---
      CALL #A_3126_MXZ02MA ;
//
//-Write outputs---
      U     #A_3126_MXZ02MA.A_3225_MXZ02.OutpRunFwd;
      =     A   1004.2;
NETWORK
TITLE ==A-3126-MXZ01MA : FAN 2
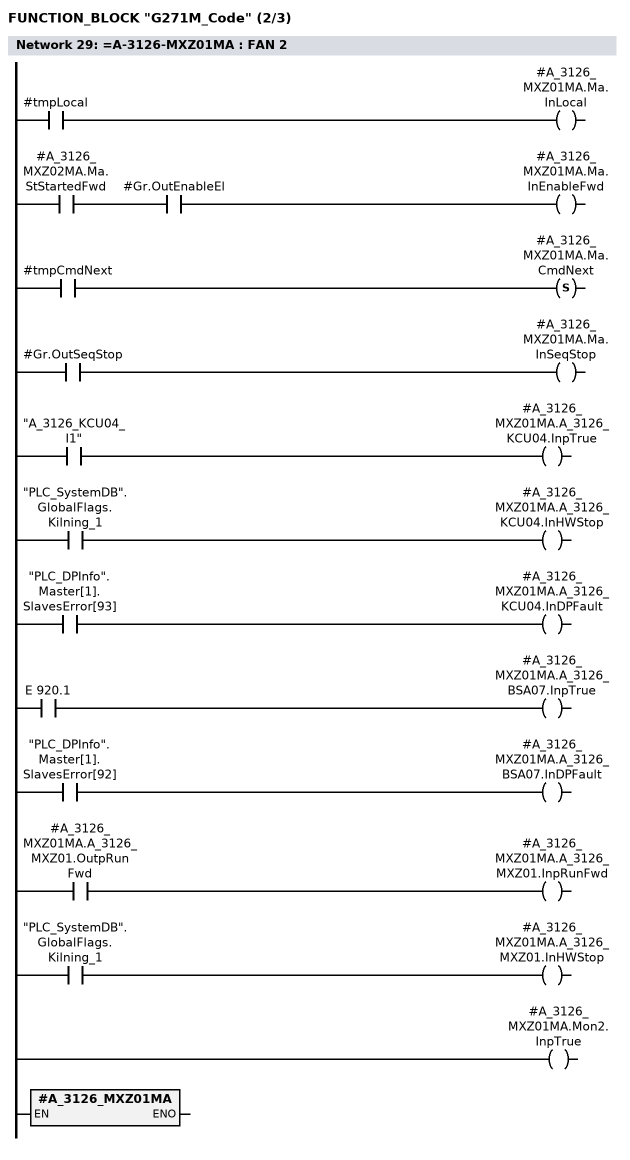

      NOP   0;
//-InLocal---
      U     #tmpLocal;
      =     #A_3126_MXZ01MA.Ma.InLocal;
//
//-Interlocking---
      U     #A_3126_MXZ02MA.Ma.StStartedFwd;
      U     #Gr.OutEnableEl;
      =     #A_3126_MXZ01MA.Ma.InEnableFwd;
//
      U     #tmpCmdNext;
      S     #A_3126_MXZ01MA.Ma.CmdNext;
//
      U     #Gr.OutSeqStop;
      =     #A_3126_MXZ01MA.Ma.InSeqStop;
//
//=Values and commands of elements===
//-=A-3126-KCU04---
//      CLR
//      S     #A_3126_MXZ01MA.A_3126_KCU04.CmdRunTimeOutTime
//-=A-3126-BSA07---
//      CLR
//      S     #A_3126_MXZ01MA.A_3126_BSA07.CmdRunTimeOutTime
//
//-Read inputs of elements---
      U     "A_3126_KCU04_I1";
      =     #A_3126_MXZ01MA.A_3126_KCU04.InpTrue;
      U     "PLC_SystemDB".GlobalFlags.Kilning_1;
      =     #A_3126_MXZ01MA.A_3126_KCU04.InHWStop;
      U     "PLC_DPInfo".Master[1].SlavesError[93];
      =     #A_3126_MXZ01MA.A_3126_KCU04.InDPFault;
      U     E    920.1;
      =     #A_3126_MXZ01MA.A_3126_BSA07.InpTrue;
      U     "PLC_DPInfo".Master[1].SlavesError[92];
      =     #A_3126_MXZ01MA.A_3126_BSA07.InDPFault;
      U     #A_3126_MXZ01MA.A_3126_MXZ01.OutpRunFwd;
      =     #A_3126_MXZ01MA.A_3126_MXZ01.InpRunFwd;
      U     "PLC_SystemDB".GlobalFlags.Kilning_1;
      =     #A_3126_MXZ01MA.A_3126_MXZ01.InHWStop;
      SET   ;
      =     #A_3126_MXZ01MA.Mon2.InpTrue;
//
//-Set Parameters---
//
//-Call object control---
      CALL #A_3126_MXZ01MA ;
//
//-Write outputs---
NETWORK
TITLE ==A-3126-TSC01_COM : FAN 2 FU KOMMUNIKATION
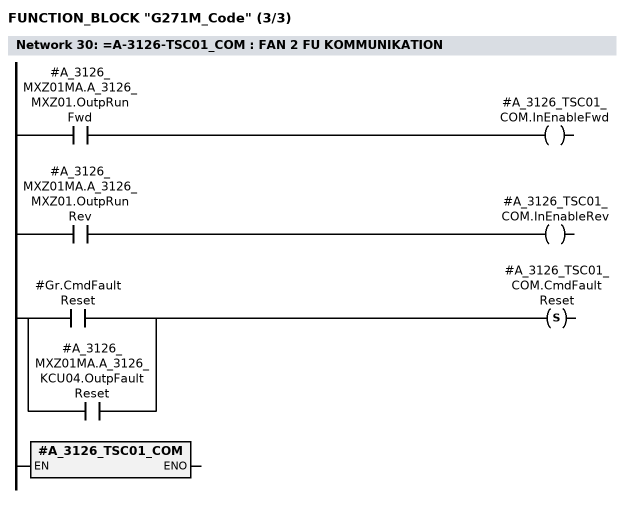

      NOP   0;
      U     #A_3126_MXZ01MA.A_3126_MXZ01.OutpRunFwd;
      =     #A_3126_TSC01_COM.InEnableFwd;
      U     #A_3126_MXZ01MA.A_3126_MXZ01.OutpRunRev;
      =     #A_3126_TSC01_COM.InEnableRev;
      U     #Gr.CmdFaultReset;
      O     #A_3126_MXZ01MA.A_3126_KCU04.OutpFaultReset;
      S     #A_3126_TSC01_COM.CmdFaultReset;
//
//
//-Read inputs---
//
//-Set Parameters---
//
//-Call object control---
      CALL #A_3126_TSC01_COM ;
//
//-Write outputs---
NETWORK
TITLE ==A-3126-TSC01_AC : ACT. CURRENT FAN 2 FU

      NOP   0;
//-InLocal---
      U     #tmpLocal;
      =     #A_3126_TSC01_AC.InLocal;
//
//-Monitoring---
      SET   ;
      =     #A_3126_TSC01_AC.InMonLL;
      CLR   ;
      =     #A_3126_TSC01_AC.InMonL;
      CLR   ;
      =     #A_3126_TSC01_AC.InMonMid;
      CLR   ;
      =     #A_3126_TSC01_AC.InMonH;
      SET   ;
      =     #A_3126_TSC01_AC.InMonHH;
//
//-Read inputs---
      L     #A_3126_TSC01_COM.Output.SetpointValue01;
      ITD   ;
      DTR   ;
      ABS   ;
      RND   ;
      T     #A_3126_TSC01_AC.InpValue;
      U     "PLC_SystemDB".GlobalFlags.Kilning_1;
      =     #A_3126_TSC01_AC.InHWStop;
//
//-Set Parameters---
//
//-Call object control---
      CALL #A_3126_TSC01_AC ;
//
//-Write outputs---
NETWORK
TITLE ==A-3126-TSC01_AF : ACT. FREQUENCY FAN 2 FU

      NOP   0;
//-InLocal---
      U     #tmpLocal;
      =     #A_3126_TSC01_AF.InLocal;
//
//-Monitoring---
      SET   ;
      =     #A_3126_TSC01_AF.InMonLL;
      CLR   ;
      =     #A_3126_TSC01_AF.InMonL;
      CLR   ;
      =     #A_3126_TSC01_AF.InMonMid;
      CLR   ;
      =     #A_3126_TSC01_AF.InMonH;
      CLR   ;
      =     #A_3126_TSC01_AF.InMonHH;
//
//-Read inputs---
      L     #A_3126_TSC01_COM.Output.SetpointValue01;
      ITD   ;
      DTR   ;
      ABS   ;
      RND   ;
      T     #A_3126_TSC01_AF.InpValue;
      U     "PLC_SystemDB".GlobalFlags.Kilning_1;
      =     #A_3126_TSC01_AF.InHWStop;
//
//-Set Parameters---
//
//-Call object control---
      CALL #A_3126_TSC01_AF ;
//
//-Write outputs---
NETWORK
TITLE ==A-3126-TSC01_AP : ACT. POWER FAN 2 FU

      NOP   0;
//-InLocal---
      U     #tmpLocal;
      =     #A_3126_TSC01_AP.InLocal;
//
//-Monitoring---
      CLR   ;
      =     #A_3126_TSC01_AP.InMonLL;
      CLR   ;
      =     #A_3126_TSC01_AP.InMonL;
      CLR   ;
      =     #A_3126_TSC01_AP.InMonMid;
      CLR   ;
      =     #A_3126_TSC01_AP.InMonH;
      CLR   ;
      =     #A_3126_TSC01_AP.InMonHH;
//
//-Read inputs---
      L     #A_3126_TSC01_COM.Output.SetpointValue01;
      ITD   ;
      DTR   ;
      ABS   ;
      RND   ;
      T     #A_3126_TSC01_AP.InpValue;
      U     "PLC_SystemDB".GlobalFlags.Kilning_1;
      =     #A_3126_TSC01_AP.InHWStop;
//
//-Set Parameters---
//
//-Call object control---
      CALL #A_3126_TSC01_AP ;
//
//-Write outputs---
NETWORK
TITLE ==A-3126-TSC01_AT : ACT. TORQUE FAN 2 FU

      NOP   0;
//-InLocal---
      U     #tmpLocal;
      =     #A_3126_TSC01_AT.InLocal;
//
//-Monitoring---
      CLR   ;
      =     #A_3126_TSC01_AT.InMonLL;
      CLR   ;
      =     #A_3126_TSC01_AT.InMonL;
      CLR   ;
      =     #A_3126_TSC01_AT.InMonMid;
      CLR   ;
      =     #A_3126_TSC01_AT.InMonH;
      CLR   ;
      =     #A_3126_TSC01_AT.InMonHH;
//
//-Read inputs---
      L     #A_3126_TSC01_COM.Output.SetpointValue01;
      ITD   ;
      DTR   ;
      ABS   ;
      RND   ;
      T     #A_3126_TSC01_AT.InpValue;
      U     "PLC_SystemDB".GlobalFlags.Kilning_1;
      =     #A_3126_TSC01_AT.InHWStop;
//
//-Set Parameters---
//
//-Call object control---
      CALL #A_3126_TSC01_AT ;
//
//-Write outputs---
NETWORK
TITLE ==A-3125-TSC01 : FAN 1 FU KOMMUNIKATION

      NOP   0;
//-InLocal---
      U     #tmpLocal;
      =     #A_3125_TSC01.InLocal;
//
//-Monitoring---
      CLR   ;
      =     #A_3125_TSC01.InMonTrue;
      CLR   ;
      =     #A_3125_TSC01.InMonFalse;
//
//-PreAlarm---
      CLR   ;
      =     #A_3125_TSC01.InPreAlarmTrue;
      CLR   ;
      =     #A_3125_TSC01.InPreAlarmFalse;
//
//-Additional commands---
//      CLR
//      S     #A_3125_TSC01.CmdRunTimeOutTime
//
//-Read inputs---
      U     "ENG_RemarkFlag";
      =     #A_3125_TSC01.InpTrue;
//
//-Set Parameters---
//
//-Call object control---
      CALL #A_3125_TSC01 ;
//
//-Write outputs---
NETWORK
TITLE ==A-3126-TSC01 : FAN 2 FU KOMMUNIKATION

      NOP   0;
//-InLocal---
      U     #tmpLocal;
      =     #A_3126_TSC01.InLocal;
//
//-Monitoring---
      CLR   ;
      =     #A_3126_TSC01.InMonTrue;
      CLR   ;
      =     #A_3126_TSC01.InMonFalse;
//
//-PreAlarm---
      CLR   ;
      =     #A_3126_TSC01.InPreAlarmTrue;
      CLR   ;
      =     #A_3126_TSC01.InPreAlarmFalse;
//
//-Additional commands---
//      CLR
//      S     #A_3126_TSC01.CmdRunTimeOutTime
//
//-Read inputs---
      U     "ENG_RemarkFlag";
      =     #A_3126_TSC01.InpTrue;
//
//-Set Parameters---
//
//-Call object control---
      CALL #A_3126_TSC01 ;
//
//-Write outputs---
NETWORK
TITLE =Test Fault
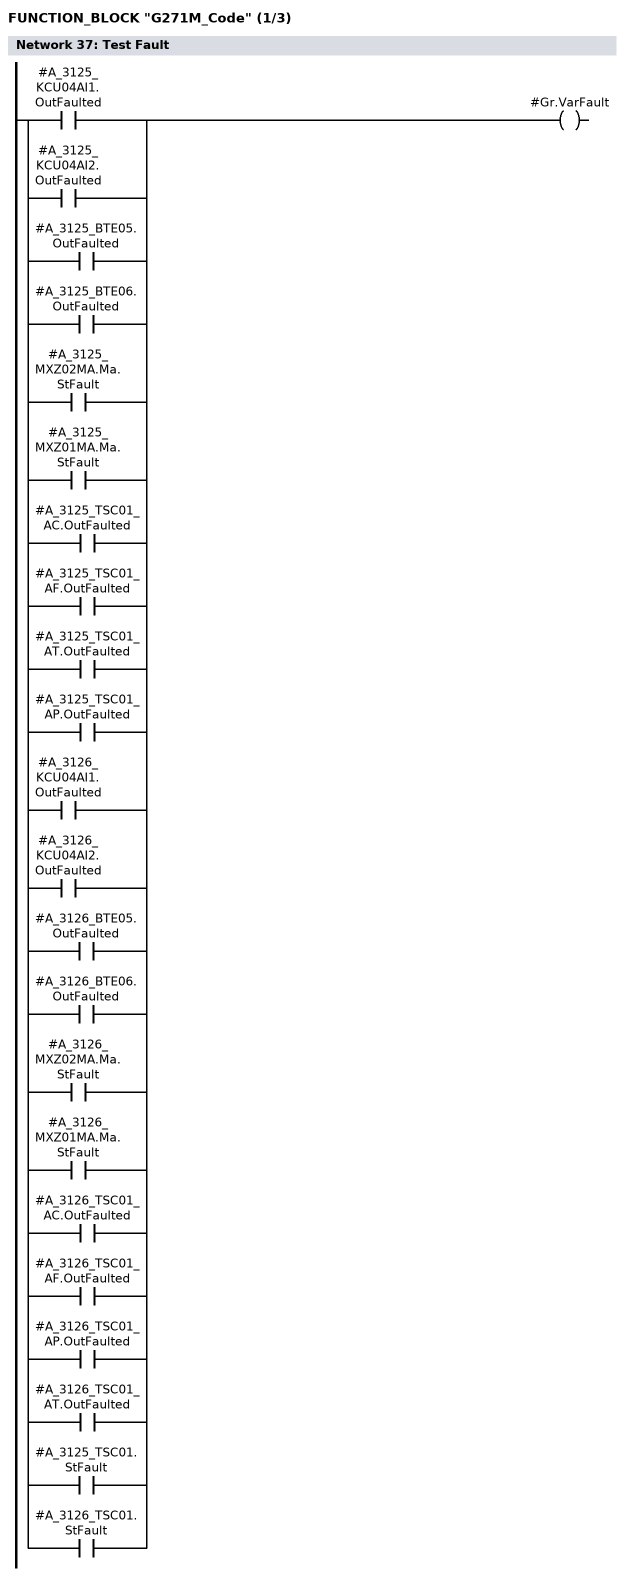

      U     #A_3125_KCU04AI1.OutFaulted;
      O     #A_3125_KCU04AI2.OutFaulted;
      O     #A_3125_BTE05.OutFaulted;
      O     #A_3125_BTE06.OutFaulted;
      O     #A_3125_MXZ02MA.Ma.StFault;
      O     #A_3125_MXZ01MA.Ma.StFault;
      O     #A_3125_TSC01_AC.OutFaulted;
      O     #A_3125_TSC01_AF.OutFaulted;
      O     #A_3125_TSC01_AT.OutFaulted;
      O     #A_3125_TSC01_AP.OutFaulted;
      O     #A_3126_KCU04AI1.OutFaulted;
      O     #A_3126_KCU04AI2.OutFaulted;
      O     #A_3126_BTE05.OutFaulted;
      O     #A_3126_BTE06.OutFaulted;
      O     #A_3126_MXZ02MA.Ma.StFault;
      O     #A_3126_MXZ01MA.Ma.StFault;
      O     #A_3126_TSC01_AC.OutFaulted;
      O     #A_3126_TSC01_AF.OutFaulted;
      O     #A_3126_TSC01_AP.OutFaulted;
      O     #A_3126_TSC01_AT.OutFaulted;
      O     #A_3125_TSC01.StFault;
      O     #A_3126_TSC01.StFault;
      =     #Gr.VarFault;
NETWORK
TITLE =Test Warning
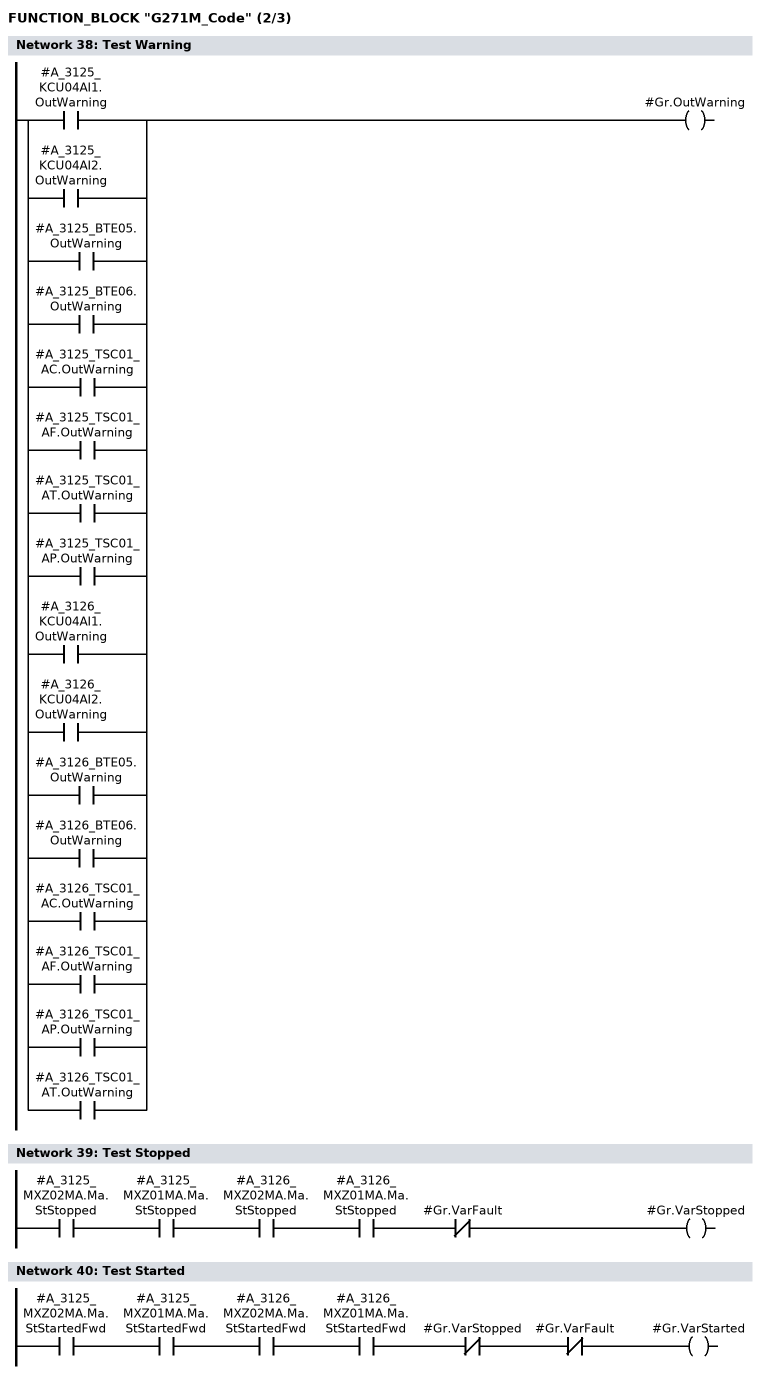

      U     #A_3125_KCU04AI1.OutWarning;
      O     #A_3125_KCU04AI2.OutWarning;
      O     #A_3125_BTE05.OutWarning;
      O     #A_3125_BTE06.OutWarning;
      O     #A_3125_TSC01_AC.OutWarning;
      O     #A_3125_TSC01_AF.OutWarning;
      O     #A_3125_TSC01_AT.OutWarning;
      O     #A_3125_TSC01_AP.OutWarning;
      O     #A_3126_KCU04AI1.OutWarning;
      O     #A_3126_KCU04AI2.OutWarning;
      O     #A_3126_BTE05.OutWarning;
      O     #A_3126_BTE06.OutWarning;
      O     #A_3126_TSC01_AC.OutWarning;
      O     #A_3126_TSC01_AF.OutWarning;
      O     #A_3126_TSC01_AP.OutWarning;
      O     #A_3126_TSC01_AT.OutWarning;
      =     #Gr.OutWarning;
NETWORK
TITLE =Test Stopped

      U     #A_3125_MXZ02MA.Ma.StStopped;
      U     #A_3125_MXZ01MA.Ma.StStopped;
      U     #A_3126_MXZ02MA.Ma.StStopped;
      U     #A_3126_MXZ01MA.Ma.StStopped;
      UN    #Gr.VarFault;
      =     #Gr.VarStopped;
NETWORK
TITLE =Test Started

      U     #A_3125_MXZ02MA.Ma.StStartedFwd;
      U     #A_3125_MXZ01MA.Ma.StStartedFwd;
      U     #A_3126_MXZ02MA.Ma.StStartedFwd;
      U     #A_3126_MXZ01MA.Ma.StStartedFwd;
      UN    #Gr.VarStopped;
      UN    #Gr.VarFault;
      =     #Gr.VarStarted;
NETWORK
TITLE =Enable Previous Group
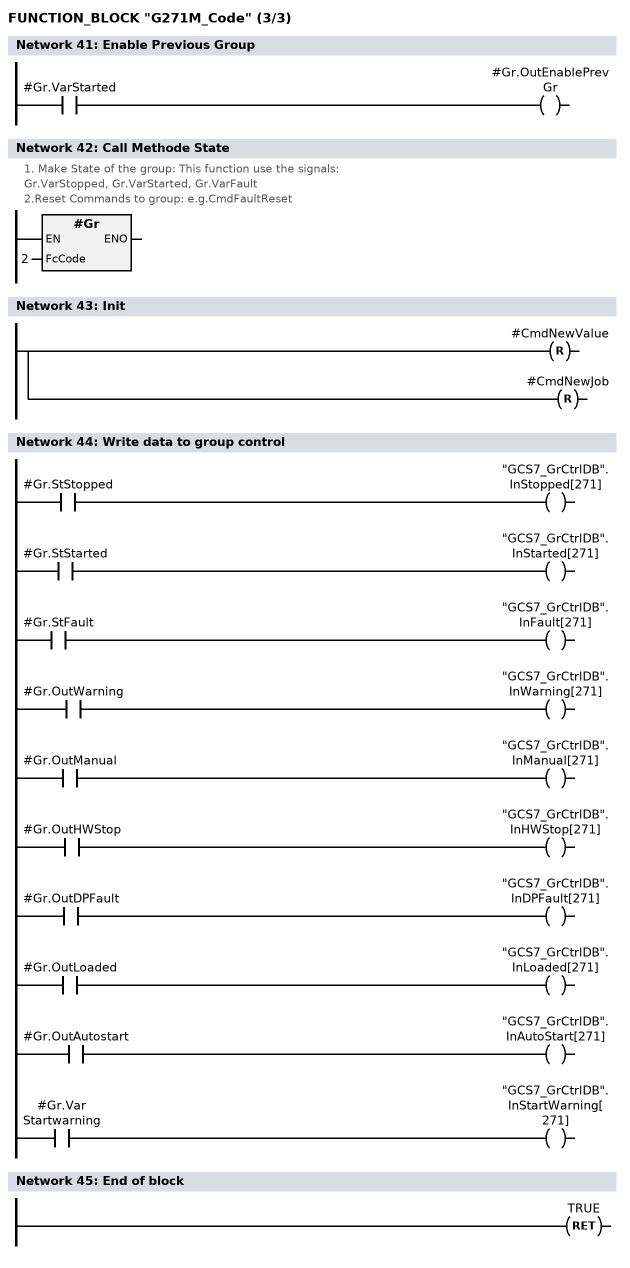

      U     #Gr.VarStarted;
      =     #Gr.OutEnablePrevGr;
NETWORK
TITLE =Call Methode State
//1. Make State of the group: This function use the signals:
//        Gr.VarStopped, Gr.VarStarted, Gr.VarFault
//2.Reset Commands to group: e.g.CmdFaultReset
      CALL #Gr (
           FcCode                   := 2);
NETWORK
TITLE =Init

      SET   ;
      R     #CmdNewValue;
      R     #CmdNewJob;
NETWORK
TITLE =Write data to group control

      U     #Gr.StStopped;
      =     "GCS7_GrCtrlDB".InStopped[271];
      U     #Gr.StStarted;
      =     "GCS7_GrCtrlDB".InStarted[271];
      U     #Gr.StFault;
      =     "GCS7_GrCtrlDB".InFault[271];
      U     #Gr.OutWarning;
      =     "GCS7_GrCtrlDB".InWarning[271];
      U     #Gr.OutManual;
      =     "GCS7_GrCtrlDB".InManual[271];
      U     #Gr.OutHWStop;
      =     "GCS7_GrCtrlDB".InHWStop[271];
      U     #Gr.OutDPFault;
      =     "GCS7_GrCtrlDB".InDPFault[271];
      U     #Gr.OutLoaded;
      =     "GCS7_GrCtrlDB".InLoaded[271];
      U     #Gr.OutAutostart;
      =     "GCS7_GrCtrlDB".InAutoStart[271];
      U     #Gr.VarStartwarning;
      =     "GCS7_GrCtrlDB".InStartWarning[271];
NETWORK
TITLE =End of block

      BE    ;
END_FUNCTION_BLOCK


DATA_BLOCK "G271M"
TITLE =DBG271M  FAN KILN 1
//COPYRIGHT:    (C) 2009  BUHLER AG, CH-9240 UZWIL, SWITZERLAND
//
//PRODUCT:      WinCoS_BIW01_09
//
//TITLE:        FAN KILN 1
//                Machine group DB
//                Maschinengruppen-DB
//
//-------------------------------------------------------------------------
//
//IDENT:        AUTHOR:             DEPT:             DATE:
//
//P01_DB371.1.0 K.Renz              CSB41             20.Mai.2010
//              1st Release
//
//-------------------------------------------------------------------------
//
//PURPOSE:
//
//MANUAL :
//
//RESTRICTIONS:
//
//-------------------------------------------------------------------------
AUTHOR : KR
FAMILY : USW
NAME : DBG271M
VERSION : 0.0

"G271M_Code"
BEGIN
   Gr.FcCode := 0;
   Gr.Spare2 := 0;
   Gr.Spare4 := 0;
   Gr.Spare6 := 0;
   Gr.OutEmptyingTime := 0;
   Gr.ChangeBit.spare := B#16#0;
   Gr.ChangeBit.CBit1 := FALSE;
   Gr.ChangeBit.CBit2 := FALSE;
   Gr.ChangeBit.CBit3 := FALSE;
   Gr.ChangeBit.CBit4 := FALSE;
   Gr.StCode := 0;
   Gr.InEnableGr := FALSE;
   Gr.CmdContinue := FALSE;
   Gr.CmdRestartIdling := FALSE;
   Gr.InReleaseEmptyingTime := FALSE;
   Gr.InFeeding := FALSE;
   Gr.InOutAutostartMan := FALSE;
   Gr.InPreStart := FALSE;
   Gr.CmdManualOff := FALSE;
   Gr.CmdOff := FALSE;
   Gr.CmdOn := FALSE;
   Gr.CmdNext := FALSE;
   Gr.CmdFaultReset := FALSE;
   Gr.InOccupied := FALSE;
   Gr.InManual := FALSE;
   Gr.InLoadedSec := FALSE;
   Gr.InSeqStop := FALSE;
   Gr.ModePassive := FALSE;
   Gr.ModeActive := FALSE;
   Gr.ModeIdling := FALSE;
   Gr.spare163 := FALSE;
   Gr.spare164 := FALSE;
   Gr.spare165 := FALSE;
   Gr.spare166 := FALSE;
   Gr.spare167 := FALSE;
   Gr.StStopped := FALSE;
   Gr.StStarting := FALSE;
   Gr.StStarted := FALSE;
   Gr.StStopping := FALSE;
   Gr.StFault := FALSE;
   Gr.OutLoaded := FALSE;
   Gr.OutWarning := FALSE;
   Gr.OutFeeding := FALSE;
   Gr.OutEnableEl := FALSE;
   Gr.OutEnable1 := FALSE;
   Gr.OutHWStop := FALSE;
   Gr.OutDPFault := FALSE;
   Gr.OutAutostart := FALSE;
   Gr.OutManual := FALSE;
   Gr.OutHornOn := FALSE;
   Gr.OutEnablePrevGr := FALSE;
   Gr.VarStopped := FALSE;
   Gr.VarStarted := FALSE;
   Gr.VarFault := FALSE;
   Gr.VarStartwarning := FALSE;
   Gr.VarFlag1s := FALSE;
   Gr.OutEmptyingTimeDone := FALSE;
   Gr.OutNewWay := FALSE;
   Gr.OutSeqStop := FALSE;
   Gr.OutIdlingTime := 0;
   Gr.InCodePreselect := 0;
   Gr.InLine := 0;
   Gr.InCode := 0;
   Gr.OutCode := 0;
   Gr.Par.ParObjectNo := 27100;
   Gr.Par.ParMgr := TRUE;
   Gr.Par.ParWgr := FALSE;
   Gr.Par.ParGgr := FALSE;
   Gr.Par.ParHornCode := 10;
   Gr.Par.ParIdling := 2;
   Gr.Par.ParEmptyingTime := 0;
   Gr.Par.Para1_0 := FALSE;
   Gr.Par.Para1_1 := FALSE;
   Gr.Par.Para1_2 := FALSE;
   Gr.Par.Para1_3 := FALSE;
   Gr.Par.Para1_4 := FALSE;
   Gr.Par.Para1_5 := FALSE;
   Gr.Par.Para1_6 := FALSE;
   Gr.Par.Para1_7 := FALSE;
   Gr.Par.Para1_8 := FALSE;
   Gr.Par.Para1_9 := FALSE;
   Gr.Par.Para1_10 := FALSE;
   Gr.Par.Para1_11 := FALSE;
   Gr.Par.Para1_12 := FALSE;
   Gr.Par.Para1_13 := FALSE;
   Gr.Par.Para1_14 := FALSE;
   Gr.Par.Para1_15 := FALSE;
   Gr.Par.Para2 := 0;
   Gr.Par.Para3 := 0;
   Gr.Par.Para4 := 0;
   Gr.Par.Para5 := 0;
   InOutValue1 := L#0;
   InOutValue2 := L#0;
   OutWayConflict := FALSE;
   OutSelectionOk := FALSE;
   CmdNewValue := FALSE;
   CmdNewJob := FALSE;
   OutCodeOK := FALSE;
   InEndOfJob := FALSE;
   staWayOk := FALSE;
   EdgeStartRelease := FALSE;
   USW8 := FALSE;
   USW9 := FALSE;
   USW10 := FALSE;
   USW11 := FALSE;
   USW12 := FALSE;
   USW13 := FALSE;
   USW14 := FALSE;
   USW15 := FALSE;
   A_3125_KCU04AI1.StCode := 0;
   A_3125_KCU04AI1.InMonLL := FALSE;
   A_3125_KCU04AI1.InMonL := FALSE;
   A_3125_KCU04AI1.InMonMid := FALSE;
   A_3125_KCU04AI1.InMonH := FALSE;
   A_3125_KCU04AI1.InMonHH := FALSE;
   A_3125_KCU04AI1.spare0205 := FALSE;
   A_3125_KCU04AI1.InpFaultAI := FALSE;
   A_3125_KCU04AI1.InpFaultDev := FALSE;
   A_3125_KCU04AI1.InHWStop := FALSE;
   A_3125_KCU04AI1.InDPFault := FALSE;
   A_3125_KCU04AI1.InDisable := FALSE;
   A_3125_KCU04AI1.CmdFaultReset := FALSE;
   A_3125_KCU04AI1.InLocal := FALSE;
   A_3125_KCU04AI1.spare0305 := FALSE;
   A_3125_KCU04AI1.InReport := FALSE;
   A_3125_KCU04AI1.spare0307 := FALSE;
   A_3125_KCU04AI1.OutLL := FALSE;
   A_3125_KCU04AI1.OutL := FALSE;
   A_3125_KCU04AI1.OutH := FALSE;
   A_3125_KCU04AI1.OutHH := FALSE;
   A_3125_KCU04AI1.OutOverflow := FALSE;
   A_3125_KCU04AI1.spare0405 := FALSE;
   A_3125_KCU04AI1.OutFaultAI := FALSE;
   A_3125_KCU04AI1.spare0407 := FALSE;
   A_3125_KCU04AI1.StLL := FALSE;
   A_3125_KCU04AI1.StL := FALSE;
   A_3125_KCU04AI1.StMid := FALSE;
   A_3125_KCU04AI1.StH := FALSE;
   A_3125_KCU04AI1.StHH := FALSE;
   A_3125_KCU04AI1.StFaultAI := FALSE;
   A_3125_KCU04AI1.OutWarning := FALSE;
   A_3125_KCU04AI1.OutFaulted := FALSE;
   A_3125_KCU04AI1.InpValue := 0;
   A_3125_KCU04AI1.OutValuePc := 0;
   A_3125_KCU04AI1.OutValueUnits := L#0;
   A_3125_KCU04AI1.Msg.WarningDoneLL := FALSE;
   A_3125_KCU04AI1.Msg.WarningDoneL := FALSE;
   A_3125_KCU04AI1.Msg.WarningDoneMid := FALSE;
   A_3125_KCU04AI1.Msg.WarningDoneH := FALSE;
   A_3125_KCU04AI1.Msg.WarningDoneHH := FALSE;
   A_3125_KCU04AI1.Msg.FaultDoneLL := FALSE;
   A_3125_KCU04AI1.Msg.FaultDoneL := FALSE;
   A_3125_KCU04AI1.Msg.FaultDoneMid := FALSE;
   A_3125_KCU04AI1.Msg.FaultDoneH := FALSE;
   A_3125_KCU04AI1.Msg.FaultDoneHH := FALSE;
   A_3125_KCU04AI1.Msg.FaultDoneDev := FALSE;
   A_3125_KCU04AI1.Msg.FaultDoneAI := FALSE;
   A_3125_KCU04AI1.OutAlarmNrLog := 0;
   A_3125_KCU04AI1.Par.ParObjectNo := 27101;
   A_3125_KCU04AI1.Par.ParMsgType := 7252;
   A_3125_KCU04AI1.Par.ParHornCode := 10;
   A_3125_KCU04AI1.Par.ParLogOff := FALSE;
   A_3125_KCU04AI1.Par.ParSpare0401 := FALSE;
   A_3125_KCU04AI1.Par.ParValueByUser := FALSE;
   A_3125_KCU04AI1.Par.ParLimitsPc := TRUE;
   A_3125_KCU04AI1.Par.ParWago := FALSE;
   A_3125_KCU04AI1.Par.ParNoHornByWarning := FALSE;
   A_3125_KCU04AI1.Par.ParWarningLL := FALSE;
   A_3125_KCU04AI1.Par.ParWarningL := FALSE;
   A_3125_KCU04AI1.Par.ParWarningMid := FALSE;
   A_3125_KCU04AI1.Par.ParWarningH := TRUE;
   A_3125_KCU04AI1.Par.ParWarningHH := FALSE;
   A_3125_KCU04AI1.Par.ParPreAlarmLL := FALSE;
   A_3125_KCU04AI1.Par.ParPreAlarmL := FALSE;
   A_3125_KCU04AI1.Par.ParPreAlarmMid := FALSE;
   A_3125_KCU04AI1.Par.ParPreAlarmH := FALSE;
   A_3125_KCU04AI1.Par.ParPreAlarmHH := FALSE;
   A_3125_KCU04AI1.Par.ParUnitsByZeroDigit := L#0;
   A_3125_KCU04AI1.Par.ParUnitsByMaxDigit := L#2000;
   A_3125_KCU04AI1.Par.ParUnitsBy100Pc := L#10000;
   A_3125_KCU04AI1.Par.ParLimitLL := L#-1;
   A_3125_KCU04AI1.Par.ParLimitL := L#0;
   A_3125_KCU04AI1.Par.ParLimitH := L#3150;
   A_3125_KCU04AI1.Par.ParLimitHH := L#3550;
   A_3125_KCU04AI1.Par.ParMonTimeLL := 0;
   A_3125_KCU04AI1.Par.ParMonTimeL := 0;
   A_3125_KCU04AI1.Par.ParMonTimeMid := 0;
   A_3125_KCU04AI1.Par.ParMonTimeH := 600;
   A_3125_KCU04AI1.Par.ParMonTimeHH := 0;
   A_3125_KCU04AI1.Par.ParDelayTimeDown := 10;
   A_3125_KCU04AI1.Par.ParDelayTimeUp := 10;
   A_3125_KCU04AI1.Par.ParDelayTime := 30;
   A_3125_KCU04AI1.Par.OutMonTimeLL := 0;
   A_3125_KCU04AI1.Par.OutMonTimeL := 0;
   A_3125_KCU04AI1.Par.OutMonTimeMid := 0;
   A_3125_KCU04AI1.Par.OutMonTimeH := 0;
   A_3125_KCU04AI1.Par.OutMonTimeHH := 0;
   A_3125_KCU04AI1.Par.OutDelayTimeDown := 0;
   A_3125_KCU04AI1.Par.OutDelayTimeUp := 0;
   A_3125_KCU04AI1.Par.OutDelayTime := 0;
   A_3125_KCU04AI1.Par.Spare66 := 0;
   A_3125_KCU04AI2.StCode := 0;
   A_3125_KCU04AI2.InMonLL := FALSE;
   A_3125_KCU04AI2.InMonL := FALSE;
   A_3125_KCU04AI2.InMonMid := FALSE;
   A_3125_KCU04AI2.InMonH := FALSE;
   A_3125_KCU04AI2.InMonHH := FALSE;
   A_3125_KCU04AI2.spare0205 := FALSE;
   A_3125_KCU04AI2.InpFaultAI := FALSE;
   A_3125_KCU04AI2.InpFaultDev := FALSE;
   A_3125_KCU04AI2.InHWStop := FALSE;
   A_3125_KCU04AI2.InDPFault := FALSE;
   A_3125_KCU04AI2.InDisable := FALSE;
   A_3125_KCU04AI2.CmdFaultReset := FALSE;
   A_3125_KCU04AI2.InLocal := FALSE;
   A_3125_KCU04AI2.spare0305 := FALSE;
   A_3125_KCU04AI2.InReport := FALSE;
   A_3125_KCU04AI2.spare0307 := FALSE;
   A_3125_KCU04AI2.OutLL := FALSE;
   A_3125_KCU04AI2.OutL := FALSE;
   A_3125_KCU04AI2.OutH := FALSE;
   A_3125_KCU04AI2.OutHH := FALSE;
   A_3125_KCU04AI2.OutOverflow := FALSE;
   A_3125_KCU04AI2.spare0405 := FALSE;
   A_3125_KCU04AI2.OutFaultAI := FALSE;
   A_3125_KCU04AI2.spare0407 := FALSE;
   A_3125_KCU04AI2.StLL := FALSE;
   A_3125_KCU04AI2.StL := FALSE;
   A_3125_KCU04AI2.StMid := FALSE;
   A_3125_KCU04AI2.StH := FALSE;
   A_3125_KCU04AI2.StHH := FALSE;
   A_3125_KCU04AI2.StFaultAI := FALSE;
   A_3125_KCU04AI2.OutWarning := FALSE;
   A_3125_KCU04AI2.OutFaulted := FALSE;
   A_3125_KCU04AI2.InpValue := 0;
   A_3125_KCU04AI2.OutValuePc := 0;
   A_3125_KCU04AI2.OutValueUnits := L#0;
   A_3125_KCU04AI2.Msg.WarningDoneLL := FALSE;
   A_3125_KCU04AI2.Msg.WarningDoneL := FALSE;
   A_3125_KCU04AI2.Msg.WarningDoneMid := FALSE;
   A_3125_KCU04AI2.Msg.WarningDoneH := FALSE;
   A_3125_KCU04AI2.Msg.WarningDoneHH := FALSE;
   A_3125_KCU04AI2.Msg.FaultDoneLL := FALSE;
   A_3125_KCU04AI2.Msg.FaultDoneL := FALSE;
   A_3125_KCU04AI2.Msg.FaultDoneMid := FALSE;
   A_3125_KCU04AI2.Msg.FaultDoneH := FALSE;
   A_3125_KCU04AI2.Msg.FaultDoneHH := FALSE;
   A_3125_KCU04AI2.Msg.FaultDoneDev := FALSE;
   A_3125_KCU04AI2.Msg.FaultDoneAI := FALSE;
   A_3125_KCU04AI2.OutAlarmNrLog := 0;
   A_3125_KCU04AI2.Par.ParObjectNo := 27102;
   A_3125_KCU04AI2.Par.ParMsgType := 7252;
   A_3125_KCU04AI2.Par.ParHornCode := 10;
   A_3125_KCU04AI2.Par.ParLogOff := FALSE;
   A_3125_KCU04AI2.Par.ParSpare0401 := FALSE;
   A_3125_KCU04AI2.Par.ParValueByUser := FALSE;
   A_3125_KCU04AI2.Par.ParLimitsPc := TRUE;
   A_3125_KCU04AI2.Par.ParWago := FALSE;
   A_3125_KCU04AI2.Par.ParNoHornByWarning := FALSE;
   A_3125_KCU04AI2.Par.ParWarningLL := FALSE;
   A_3125_KCU04AI2.Par.ParWarningL := FALSE;
   A_3125_KCU04AI2.Par.ParWarningMid := FALSE;
   A_3125_KCU04AI2.Par.ParWarningH := TRUE;
   A_3125_KCU04AI2.Par.ParWarningHH := FALSE;
   A_3125_KCU04AI2.Par.ParPreAlarmLL := FALSE;
   A_3125_KCU04AI2.Par.ParPreAlarmL := FALSE;
   A_3125_KCU04AI2.Par.ParPreAlarmMid := FALSE;
   A_3125_KCU04AI2.Par.ParPreAlarmH := FALSE;
   A_3125_KCU04AI2.Par.ParPreAlarmHH := FALSE;
   A_3125_KCU04AI2.Par.ParUnitsByZeroDigit := L#0;
   A_3125_KCU04AI2.Par.ParUnitsByMaxDigit := L#2000;
   A_3125_KCU04AI2.Par.ParUnitsBy100Pc := L#10000;
   A_3125_KCU04AI2.Par.ParLimitLL := L#-1;
   A_3125_KCU04AI2.Par.ParLimitL := L#0;
   A_3125_KCU04AI2.Par.ParLimitH := L#3150;
   A_3125_KCU04AI2.Par.ParLimitHH := L#3550;
   A_3125_KCU04AI2.Par.ParMonTimeLL := 0;
   A_3125_KCU04AI2.Par.ParMonTimeL := 0;
   A_3125_KCU04AI2.Par.ParMonTimeMid := 0;
   A_3125_KCU04AI2.Par.ParMonTimeH := 600;
   A_3125_KCU04AI2.Par.ParMonTimeHH := 0;
   A_3125_KCU04AI2.Par.ParDelayTimeDown := 10;
   A_3125_KCU04AI2.Par.ParDelayTimeUp := 10;
   A_3125_KCU04AI2.Par.ParDelayTime := 30;
   A_3125_KCU04AI2.Par.OutMonTimeLL := 0;
   A_3125_KCU04AI2.Par.OutMonTimeL := 0;
   A_3125_KCU04AI2.Par.OutMonTimeMid := 0;
   A_3125_KCU04AI2.Par.OutMonTimeH := 0;
   A_3125_KCU04AI2.Par.OutMonTimeHH := 0;
   A_3125_KCU04AI2.Par.OutDelayTimeDown := 0;
   A_3125_KCU04AI2.Par.OutDelayTimeUp := 0;
   A_3125_KCU04AI2.Par.OutDelayTime := 0;
   A_3125_KCU04AI2.Par.Spare66 := 0;
   A_3125_BTE05.StCode := 0;
   A_3125_BTE05.InMonLL := FALSE;
   A_3125_BTE05.InMonL := FALSE;
   A_3125_BTE05.InMonMid := FALSE;
   A_3125_BTE05.InMonH := FALSE;
   A_3125_BTE05.InMonHH := FALSE;
   A_3125_BTE05.spare0205 := FALSE;
   A_3125_BTE05.InpFaultAI := FALSE;
   A_3125_BTE05.InpFaultDev := FALSE;
   A_3125_BTE05.InHWStop := FALSE;
   A_3125_BTE05.InDPFault := FALSE;
   A_3125_BTE05.InDisable := FALSE;
   A_3125_BTE05.CmdFaultReset := FALSE;
   A_3125_BTE05.InLocal := FALSE;
   A_3125_BTE05.spare0305 := FALSE;
   A_3125_BTE05.InReport := FALSE;
   A_3125_BTE05.spare0307 := FALSE;
   A_3125_BTE05.OutLL := FALSE;
   A_3125_BTE05.OutL := FALSE;
   A_3125_BTE05.OutH := FALSE;
   A_3125_BTE05.OutHH := FALSE;
   A_3125_BTE05.OutOverflow := FALSE;
   A_3125_BTE05.spare0405 := FALSE;
   A_3125_BTE05.OutFaultAI := FALSE;
   A_3125_BTE05.spare0407 := FALSE;
   A_3125_BTE05.StLL := FALSE;
   A_3125_BTE05.StL := FALSE;
   A_3125_BTE05.StMid := FALSE;
   A_3125_BTE05.StH := FALSE;
   A_3125_BTE05.StHH := FALSE;
   A_3125_BTE05.StFaultAI := FALSE;
   A_3125_BTE05.OutWarning := FALSE;
   A_3125_BTE05.OutFaulted := FALSE;
   A_3125_BTE05.InpValue := 0;
   A_3125_BTE05.OutValuePc := 0;
   A_3125_BTE05.OutValueUnits := L#0;
   A_3125_BTE05.Msg.WarningDoneLL := FALSE;
   A_3125_BTE05.Msg.WarningDoneL := FALSE;
   A_3125_BTE05.Msg.WarningDoneMid := FALSE;
   A_3125_BTE05.Msg.WarningDoneH := FALSE;
   A_3125_BTE05.Msg.WarningDoneHH := FALSE;
   A_3125_BTE05.Msg.FaultDoneLL := FALSE;
   A_3125_BTE05.Msg.FaultDoneL := FALSE;
   A_3125_BTE05.Msg.FaultDoneMid := FALSE;
   A_3125_BTE05.Msg.FaultDoneH := FALSE;
   A_3125_BTE05.Msg.FaultDoneHH := FALSE;
   A_3125_BTE05.Msg.FaultDoneDev := FALSE;
   A_3125_BTE05.Msg.FaultDoneAI := FALSE;
   A_3125_BTE05.OutAlarmNrLog := 0;
   A_3125_BTE05.Par.ParObjectNo := 27103;
   A_3125_BTE05.Par.ParMsgType := 7252;
   A_3125_BTE05.Par.ParHornCode := 10;
   A_3125_BTE05.Par.ParLogOff := FALSE;
   A_3125_BTE05.Par.ParSpare0401 := FALSE;
   A_3125_BTE05.Par.ParValueByUser := FALSE;
   A_3125_BTE05.Par.ParLimitsPc := TRUE;
   A_3125_BTE05.Par.ParWago := FALSE;
   A_3125_BTE05.Par.ParNoHornByWarning := FALSE;
   A_3125_BTE05.Par.ParWarningLL := FALSE;
   A_3125_BTE05.Par.ParWarningL := FALSE;
   A_3125_BTE05.Par.ParWarningMid := FALSE;
   A_3125_BTE05.Par.ParWarningH := TRUE;
   A_3125_BTE05.Par.ParWarningHH := FALSE;
   A_3125_BTE05.Par.ParPreAlarmLL := FALSE;
   A_3125_BTE05.Par.ParPreAlarmL := FALSE;
   A_3125_BTE05.Par.ParPreAlarmMid := FALSE;
   A_3125_BTE05.Par.ParPreAlarmH := FALSE;
   A_3125_BTE05.Par.ParPreAlarmHH := FALSE;
   A_3125_BTE05.Par.ParUnitsByZeroDigit := L#0;
   A_3125_BTE05.Par.ParUnitsByMaxDigit := L#27384;
   A_3125_BTE05.Par.ParUnitsBy100Pc := L#10000;
   A_3125_BTE05.Par.ParLimitLL := L#0;
   A_3125_BTE05.Par.ParLimitL := L#2000;
   A_3125_BTE05.Par.ParLimitH := L#8000;
   A_3125_BTE05.Par.ParLimitHH := L#10000;
   A_3125_BTE05.Par.ParMonTimeLL := 0;
   A_3125_BTE05.Par.ParMonTimeL := 0;
   A_3125_BTE05.Par.ParMonTimeMid := 0;
   A_3125_BTE05.Par.ParMonTimeH := 600;
   A_3125_BTE05.Par.ParMonTimeHH := 0;
   A_3125_BTE05.Par.ParDelayTimeDown := 10;
   A_3125_BTE05.Par.ParDelayTimeUp := 10;
   A_3125_BTE05.Par.ParDelayTime := 30;
   A_3125_BTE05.Par.OutMonTimeLL := 0;
   A_3125_BTE05.Par.OutMonTimeL := 0;
   A_3125_BTE05.Par.OutMonTimeMid := 0;
   A_3125_BTE05.Par.OutMonTimeH := 0;
   A_3125_BTE05.Par.OutMonTimeHH := 0;
   A_3125_BTE05.Par.OutDelayTimeDown := 0;
   A_3125_BTE05.Par.OutDelayTimeUp := 0;
   A_3125_BTE05.Par.OutDelayTime := 0;
   A_3125_BTE05.Par.Spare66 := 0;
   A_3125_BTE06.StCode := 0;
   A_3125_BTE06.InMonLL := FALSE;
   A_3125_BTE06.InMonL := FALSE;
   A_3125_BTE06.InMonMid := FALSE;
   A_3125_BTE06.InMonH := FALSE;
   A_3125_BTE06.InMonHH := FALSE;
   A_3125_BTE06.spare0205 := FALSE;
   A_3125_BTE06.InpFaultAI := FALSE;
   A_3125_BTE06.InpFaultDev := FALSE;
   A_3125_BTE06.InHWStop := FALSE;
   A_3125_BTE06.InDPFault := FALSE;
   A_3125_BTE06.InDisable := FALSE;
   A_3125_BTE06.CmdFaultReset := FALSE;
   A_3125_BTE06.InLocal := FALSE;
   A_3125_BTE06.spare0305 := FALSE;
   A_3125_BTE06.InReport := FALSE;
   A_3125_BTE06.spare0307 := FALSE;
   A_3125_BTE06.OutLL := FALSE;
   A_3125_BTE06.OutL := FALSE;
   A_3125_BTE06.OutH := FALSE;
   A_3125_BTE06.OutHH := FALSE;
   A_3125_BTE06.OutOverflow := FALSE;
   A_3125_BTE06.spare0405 := FALSE;
   A_3125_BTE06.OutFaultAI := FALSE;
   A_3125_BTE06.spare0407 := FALSE;
   A_3125_BTE06.StLL := FALSE;
   A_3125_BTE06.StL := FALSE;
   A_3125_BTE06.StMid := FALSE;
   A_3125_BTE06.StH := FALSE;
   A_3125_BTE06.StHH := FALSE;
   A_3125_BTE06.StFaultAI := FALSE;
   A_3125_BTE06.OutWarning := FALSE;
   A_3125_BTE06.OutFaulted := FALSE;
   A_3125_BTE06.InpValue := 0;
   A_3125_BTE06.OutValuePc := 0;
   A_3125_BTE06.OutValueUnits := L#0;
   A_3125_BTE06.Msg.WarningDoneLL := FALSE;
   A_3125_BTE06.Msg.WarningDoneL := FALSE;
   A_3125_BTE06.Msg.WarningDoneMid := FALSE;
   A_3125_BTE06.Msg.WarningDoneH := FALSE;
   A_3125_BTE06.Msg.WarningDoneHH := FALSE;
   A_3125_BTE06.Msg.FaultDoneLL := FALSE;
   A_3125_BTE06.Msg.FaultDoneL := FALSE;
   A_3125_BTE06.Msg.FaultDoneMid := FALSE;
   A_3125_BTE06.Msg.FaultDoneH := FALSE;
   A_3125_BTE06.Msg.FaultDoneHH := FALSE;
   A_3125_BTE06.Msg.FaultDoneDev := FALSE;
   A_3125_BTE06.Msg.FaultDoneAI := FALSE;
   A_3125_BTE06.OutAlarmNrLog := 0;
   A_3125_BTE06.Par.ParObjectNo := 27104;
   A_3125_BTE06.Par.ParMsgType := 7252;
   A_3125_BTE06.Par.ParHornCode := 10;
   A_3125_BTE06.Par.ParLogOff := FALSE;
   A_3125_BTE06.Par.ParSpare0401 := FALSE;
   A_3125_BTE06.Par.ParValueByUser := FALSE;
   A_3125_BTE06.Par.ParLimitsPc := TRUE;
   A_3125_BTE06.Par.ParWago := FALSE;
   A_3125_BTE06.Par.ParNoHornByWarning := FALSE;
   A_3125_BTE06.Par.ParWarningLL := FALSE;
   A_3125_BTE06.Par.ParWarningL := FALSE;
   A_3125_BTE06.Par.ParWarningMid := FALSE;
   A_3125_BTE06.Par.ParWarningH := TRUE;
   A_3125_BTE06.Par.ParWarningHH := FALSE;
   A_3125_BTE06.Par.ParPreAlarmLL := FALSE;
   A_3125_BTE06.Par.ParPreAlarmL := FALSE;
   A_3125_BTE06.Par.ParPreAlarmMid := FALSE;
   A_3125_BTE06.Par.ParPreAlarmH := FALSE;
   A_3125_BTE06.Par.ParPreAlarmHH := FALSE;
   A_3125_BTE06.Par.ParUnitsByZeroDigit := L#0;
   A_3125_BTE06.Par.ParUnitsByMaxDigit := L#27384;
   A_3125_BTE06.Par.ParUnitsBy100Pc := L#10000;
   A_3125_BTE06.Par.ParLimitLL := L#0;
   A_3125_BTE06.Par.ParLimitL := L#2000;
   A_3125_BTE06.Par.ParLimitH := L#8000;
   A_3125_BTE06.Par.ParLimitHH := L#10000;
   A_3125_BTE06.Par.ParMonTimeLL := 0;
   A_3125_BTE06.Par.ParMonTimeL := 0;
   A_3125_BTE06.Par.ParMonTimeMid := 0;
   A_3125_BTE06.Par.ParMonTimeH := 600;
   A_3125_BTE06.Par.ParMonTimeHH := 0;
   A_3125_BTE06.Par.ParDelayTimeDown := 10;
   A_3125_BTE06.Par.ParDelayTimeUp := 10;
   A_3125_BTE06.Par.ParDelayTime := 30;
   A_3125_BTE06.Par.OutMonTimeLL := 0;
   A_3125_BTE06.Par.OutMonTimeL := 0;
   A_3125_BTE06.Par.OutMonTimeMid := 0;
   A_3125_BTE06.Par.OutMonTimeH := 0;
   A_3125_BTE06.Par.OutMonTimeHH := 0;
   A_3125_BTE06.Par.OutDelayTimeDown := 0;
   A_3125_BTE06.Par.OutDelayTimeUp := 0;
   A_3125_BTE06.Par.OutDelayTime := 0;
   A_3125_BTE06.Par.Spare66 := 0;
   A_3125_MXZ01MA.Ma.StCode := 0;
   A_3125_MXZ01MA.Ma.InEnableRev := FALSE;
   A_3125_MXZ01MA.Ma.InEnableFwd := FALSE;
   A_3125_MXZ01MA.Ma.InOverrideHLOutlet := FALSE;
   A_3125_MXZ01MA.Ma.spare0203 := FALSE;
   A_3125_MXZ01MA.Ma.OutEdgeFaultReset := FALSE;
   A_3125_MXZ01MA.Ma.OutFaultResetFcttst := FALSE;
   A_3125_MXZ01MA.Ma.InpControlEBM := FALSE;
   A_3125_MXZ01MA.Ma.InpLocked := FALSE;
   A_3125_MXZ01MA.Ma.CmdOff := FALSE;
   A_3125_MXZ01MA.Ma.CmdOn := FALSE;
   A_3125_MXZ01MA.Ma.CmdNext := FALSE;
   A_3125_MXZ01MA.Ma.CmdFaultReset := FALSE;
   A_3125_MXZ01MA.Ma.InLocal := FALSE;
   A_3125_MXZ01MA.Ma.InManual := FALSE;
   A_3125_MXZ01MA.Ma.CmdTestEBM := FALSE;
   A_3125_MXZ01MA.Ma.InSeqStop := FALSE;
   A_3125_MXZ01MA.Ma.OutWarning := FALSE;
   A_3125_MXZ01MA.Ma.InfBMTopOk := FALSE;
   A_3125_MXZ01MA.Ma.InfBMBottomOk := FALSE;
   A_3125_MXZ01MA.Ma.InfSMOk := FALSE;
   A_3125_MXZ01MA.Ma.OutpFcttst_BM_Top := FALSE;
   A_3125_MXZ01MA.Ma.OutpFcttst_BM_Bottom := FALSE;
   A_3125_MXZ01MA.Ma.OutpFcttst_SM := FALSE;
   A_3125_MXZ01MA.Ma.OutpFaultReset := FALSE;
   A_3125_MXZ01MA.Ma.StStopped := FALSE;
   A_3125_MXZ01MA.Ma.StStarting := FALSE;
   A_3125_MXZ01MA.Ma.StStartedFwd := FALSE;
   A_3125_MXZ01MA.Ma.StStopping := FALSE;
   A_3125_MXZ01MA.Ma.StFault := FALSE;
   A_3125_MXZ01MA.Ma.StStartedRev := FALSE;
   A_3125_MXZ01MA.Ma.StLocked := FALSE;
   A_3125_MXZ01MA.Ma.OutTestTime := 0;
   A_3125_MXZ01MA.Ma.Par.ParObjectNo := 27105;
   A_3125_MXZ01MA.Ma.Par.ParWithMon1 := TRUE;
   A_3125_MXZ01MA.Ma.Par.ParWithMon3 := FALSE;
   A_3125_MXZ01MA.Ma.Par.ParWithMon4 := TRUE;
   A_3125_MXZ01MA.Ma.Par.ParWithMon5 := FALSE;
   A_3125_MXZ01MA.Ma.Par.ParWithMon6 := FALSE;
   A_3125_MXZ01MA.Ma.Par.ParMon1IsHL := FALSE;
   A_3125_MXZ01MA.Ma.Par.ParMon1IsLS := TRUE;
   A_3125_MXZ01MA.Ma.Par.ParMon1StopByFault := TRUE;
   A_3125_MXZ01MA.Ma.Par.ParMon2IsLS := FALSE;
   A_3125_MXZ01MA.Ma.Par.ParMon3IsLS := FALSE;
   A_3125_MXZ01MA.Ma.Par.ParMon4AsWarning := FALSE;
   A_3125_MXZ01MA.Ma.Par.ParMon4StopByFault := TRUE;
   A_3125_MXZ01MA.Ma.Par.ParMon4IsLS := FALSE;
   A_3125_MXZ01MA.Ma.Par.ParEBM := FALSE;
   A_3125_MXZ01MA.Ma.Par.ParMon4IsSM := TRUE;
   A_3125_MXZ01MA.A_3125_KCU04.StCode := 0;
   A_3125_MXZ01MA.A_3125_KCU04.InMonTrue := FALSE;
   A_3125_MXZ01MA.A_3125_KCU04.InMonFalse := FALSE;
   A_3125_MXZ01MA.A_3125_KCU04.InPreAlarmTrue := FALSE;
   A_3125_MXZ01MA.A_3125_KCU04.InPreAlarmFalse := FALSE;
   A_3125_MXZ01MA.A_3125_KCU04.InStopTrueTime := FALSE;
   A_3125_MXZ01MA.A_3125_KCU04.InStopFalseTime := FALSE;
   A_3125_MXZ01MA.A_3125_KCU04.InpTrue := FALSE;
   A_3125_MXZ01MA.A_3125_KCU04.InpFaultDev := FALSE;
   A_3125_MXZ01MA.A_3125_KCU04.CmdRstTrueTime := FALSE;
   A_3125_MXZ01MA.A_3125_KCU04.CmdRstFalseTime := FALSE;
   A_3125_MXZ01MA.A_3125_KCU04.CmdRunTimeoutTime := FALSE;
   A_3125_MXZ01MA.A_3125_KCU04.CmdFaultReset := FALSE;
   A_3125_MXZ01MA.A_3125_KCU04.InLocal := FALSE;
   A_3125_MXZ01MA.A_3125_KCU04.spare0305 := FALSE;
   A_3125_MXZ01MA.A_3125_KCU04.InReport := FALSE;
   A_3125_MXZ01MA.A_3125_KCU04.OutTimeoutTime := FALSE;
   A_3125_MXZ01MA.A_3125_KCU04.InHWStop := FALSE;
   A_3125_MXZ01MA.A_3125_KCU04.InDPFault := FALSE;
   A_3125_MXZ01MA.A_3125_KCU04.OutPreAlarmTrue := FALSE;
   A_3125_MXZ01MA.A_3125_KCU04.OutPreAlarmFalse := FALSE;
   A_3125_MXZ01MA.A_3125_KCU04.OutFlagPos := FALSE;
   A_3125_MXZ01MA.A_3125_KCU04.OutFlagNeg := FALSE;
   A_3125_MXZ01MA.A_3125_KCU04.OutpFaultReset := FALSE;
   A_3125_MXZ01MA.A_3125_KCU04.OutTrue := FALSE;
   A_3125_MXZ01MA.A_3125_KCU04.StFalse := FALSE;
   A_3125_MXZ01MA.A_3125_KCU04.StCtoTrue := FALSE;
   A_3125_MXZ01MA.A_3125_KCU04.StTrue := FALSE;
   A_3125_MXZ01MA.A_3125_KCU04.StCtoFalse := FALSE;
   A_3125_MXZ01MA.A_3125_KCU04.StFault := FALSE;
   A_3125_MXZ01MA.A_3125_KCU04.OutAlarmNrLog := 0;
   A_3125_MXZ01MA.A_3125_KCU04.Par.ParObjectNo := 27106;
   A_3125_MXZ01MA.A_3125_KCU04.Par.ParMsgType := 7154;
   A_3125_MXZ01MA.A_3125_KCU04.Par.ParHornCode := 10;
   A_3125_MXZ01MA.A_3125_KCU04.Par.ParLogOff := FALSE;
   A_3125_MXZ01MA.A_3125_KCU04.Par.spare0401 := FALSE;
   A_3125_MXZ01MA.A_3125_KCU04.Par.Par2WorkingCond := FALSE;
   A_3125_MXZ01MA.A_3125_KCU04.Par.ParFaultRetry := FALSE;
   A_3125_MXZ01MA.A_3125_KCU04.Par.ParBinLevel := FALSE;
   A_3125_MXZ01MA.A_3125_KCU04.Par.ParDelayChange := 20;
   A_3125_MXZ01MA.A_3125_KCU04.Par.ParDelayTrue := 10;
   A_3125_MXZ01MA.A_3125_KCU04.Par.ParDelayFalse := 0;
   A_3125_MXZ01MA.A_3125_KCU04.Par.ParTimeoutTrue := 0;
   A_3125_MXZ01MA.A_3125_KCU04.Par.ParTimeoutFalse := 0;
   A_3125_MXZ01MA.A_3125_KCU04.Par.OutMonTime := 0;
   A_3125_MXZ01MA.A_3125_KCU04.Par.OutTransitionTime := 0;
   A_3125_MXZ01MA.A_3125_KCU04.Par.OutMonTrue := FALSE;
   A_3125_MXZ01MA.A_3125_KCU04.Par.OutMonFalse := FALSE;
   A_3125_MXZ01MA.A_3125_KCU04.Par.OutFlagFaultDev := FALSE;
   A_3125_MXZ01MA.A_3125_KCU04.Par.OutDelayTime := 0;
   A_3125_MXZ01MA.Mon2.StCode := 0;
   A_3125_MXZ01MA.Mon2.InMonTrue := FALSE;
   A_3125_MXZ01MA.Mon2.InMonFalse := FALSE;
   A_3125_MXZ01MA.Mon2.InPreAlarmTrue := FALSE;
   A_3125_MXZ01MA.Mon2.InPreAlarmFalse := FALSE;
   A_3125_MXZ01MA.Mon2.InStopTrueTime := FALSE;
   A_3125_MXZ01MA.Mon2.InStopFalseTime := FALSE;
   A_3125_MXZ01MA.Mon2.InpTrue := FALSE;
   A_3125_MXZ01MA.Mon2.InpFaultDev := FALSE;
   A_3125_MXZ01MA.Mon2.CmdRstTrueTime := FALSE;
   A_3125_MXZ01MA.Mon2.CmdRstFalseTime := FALSE;
   A_3125_MXZ01MA.Mon2.CmdRunTimeoutTime := FALSE;
   A_3125_MXZ01MA.Mon2.CmdFaultReset := FALSE;
   A_3125_MXZ01MA.Mon2.InLocal := FALSE;
   A_3125_MXZ01MA.Mon2.spare0305 := FALSE;
   A_3125_MXZ01MA.Mon2.InReport := FALSE;
   A_3125_MXZ01MA.Mon2.OutTimeoutTime := FALSE;
   A_3125_MXZ01MA.Mon2.InHWStop := FALSE;
   A_3125_MXZ01MA.Mon2.InDPFault := FALSE;
   A_3125_MXZ01MA.Mon2.OutPreAlarmTrue := FALSE;
   A_3125_MXZ01MA.Mon2.OutPreAlarmFalse := FALSE;
   A_3125_MXZ01MA.Mon2.OutFlagPos := FALSE;
   A_3125_MXZ01MA.Mon2.OutFlagNeg := FALSE;
   A_3125_MXZ01MA.Mon2.OutpFaultReset := FALSE;
   A_3125_MXZ01MA.Mon2.OutTrue := FALSE;
   A_3125_MXZ01MA.Mon2.StFalse := FALSE;
   A_3125_MXZ01MA.Mon2.StCtoTrue := FALSE;
   A_3125_MXZ01MA.Mon2.StTrue := FALSE;
   A_3125_MXZ01MA.Mon2.StCtoFalse := FALSE;
   A_3125_MXZ01MA.Mon2.StFault := FALSE;
   A_3125_MXZ01MA.Mon2.OutAlarmNrLog := 0;
   A_3125_MXZ01MA.Mon2.Par.ParObjectNo := 0;
   A_3125_MXZ01MA.Mon2.Par.ParMsgType := 0;
   A_3125_MXZ01MA.Mon2.Par.ParHornCode := 0;
   A_3125_MXZ01MA.Mon2.Par.ParLogOff := FALSE;
   A_3125_MXZ01MA.Mon2.Par.spare0401 := FALSE;
   A_3125_MXZ01MA.Mon2.Par.Par2WorkingCond := FALSE;
   A_3125_MXZ01MA.Mon2.Par.ParFaultRetry := FALSE;
   A_3125_MXZ01MA.Mon2.Par.ParBinLevel := FALSE;
   A_3125_MXZ01MA.Mon2.Par.ParDelayChange := 0;
   A_3125_MXZ01MA.Mon2.Par.ParDelayTrue := 0;
   A_3125_MXZ01MA.Mon2.Par.ParDelayFalse := 0;
   A_3125_MXZ01MA.Mon2.Par.ParTimeoutTrue := 0;
   A_3125_MXZ01MA.Mon2.Par.ParTimeoutFalse := 0;
   A_3125_MXZ01MA.Mon2.Par.OutMonTime := 0;
   A_3125_MXZ01MA.Mon2.Par.OutTransitionTime := 0;
   A_3125_MXZ01MA.Mon2.Par.OutMonTrue := FALSE;
   A_3125_MXZ01MA.Mon2.Par.OutMonFalse := FALSE;
   A_3125_MXZ01MA.Mon2.Par.OutFlagFaultDev := FALSE;
   A_3125_MXZ01MA.Mon2.Par.OutDelayTime := 0;
   A_3125_MXZ01MA.Mon3.StCode := 0;
   A_3125_MXZ01MA.Mon3.InMonTrue := FALSE;
   A_3125_MXZ01MA.Mon3.InMonFalse := FALSE;
   A_3125_MXZ01MA.Mon3.InPreAlarmTrue := FALSE;
   A_3125_MXZ01MA.Mon3.InPreAlarmFalse := FALSE;
   A_3125_MXZ01MA.Mon3.InStopTrueTime := FALSE;
   A_3125_MXZ01MA.Mon3.InStopFalseTime := FALSE;
   A_3125_MXZ01MA.Mon3.InpTrue := FALSE;
   A_3125_MXZ01MA.Mon3.InpFaultDev := FALSE;
   A_3125_MXZ01MA.Mon3.CmdRstTrueTime := FALSE;
   A_3125_MXZ01MA.Mon3.CmdRstFalseTime := FALSE;
   A_3125_MXZ01MA.Mon3.CmdRunTimeoutTime := FALSE;
   A_3125_MXZ01MA.Mon3.CmdFaultReset := FALSE;
   A_3125_MXZ01MA.Mon3.InLocal := FALSE;
   A_3125_MXZ01MA.Mon3.spare0305 := FALSE;
   A_3125_MXZ01MA.Mon3.InReport := FALSE;
   A_3125_MXZ01MA.Mon3.OutTimeoutTime := FALSE;
   A_3125_MXZ01MA.Mon3.InHWStop := FALSE;
   A_3125_MXZ01MA.Mon3.InDPFault := FALSE;
   A_3125_MXZ01MA.Mon3.OutPreAlarmTrue := FALSE;
   A_3125_MXZ01MA.Mon3.OutPreAlarmFalse := FALSE;
   A_3125_MXZ01MA.Mon3.OutFlagPos := FALSE;
   A_3125_MXZ01MA.Mon3.OutFlagNeg := FALSE;
   A_3125_MXZ01MA.Mon3.OutpFaultReset := FALSE;
   A_3125_MXZ01MA.Mon3.OutTrue := FALSE;
   A_3125_MXZ01MA.Mon3.StFalse := FALSE;
   A_3125_MXZ01MA.Mon3.StCtoTrue := FALSE;
   A_3125_MXZ01MA.Mon3.StTrue := FALSE;
   A_3125_MXZ01MA.Mon3.StCtoFalse := FALSE;
   A_3125_MXZ01MA.Mon3.StFault := FALSE;
   A_3125_MXZ01MA.Mon3.OutAlarmNrLog := 0;
   A_3125_MXZ01MA.Mon3.Par.ParObjectNo := 0;
   A_3125_MXZ01MA.Mon3.Par.ParMsgType := 0;
   A_3125_MXZ01MA.Mon3.Par.ParHornCode := 0;
   A_3125_MXZ01MA.Mon3.Par.ParLogOff := FALSE;
   A_3125_MXZ01MA.Mon3.Par.spare0401 := FALSE;
   A_3125_MXZ01MA.Mon3.Par.Par2WorkingCond := FALSE;
   A_3125_MXZ01MA.Mon3.Par.ParFaultRetry := FALSE;
   A_3125_MXZ01MA.Mon3.Par.ParBinLevel := FALSE;
   A_3125_MXZ01MA.Mon3.Par.ParDelayChange := 0;
   A_3125_MXZ01MA.Mon3.Par.ParDelayTrue := 0;
   A_3125_MXZ01MA.Mon3.Par.ParDelayFalse := 0;
   A_3125_MXZ01MA.Mon3.Par.ParTimeoutTrue := 0;
   A_3125_MXZ01MA.Mon3.Par.ParTimeoutFalse := 0;
   A_3125_MXZ01MA.Mon3.Par.OutMonTime := 0;
   A_3125_MXZ01MA.Mon3.Par.OutTransitionTime := 0;
   A_3125_MXZ01MA.Mon3.Par.OutMonTrue := FALSE;
   A_3125_MXZ01MA.Mon3.Par.OutMonFalse := FALSE;
   A_3125_MXZ01MA.Mon3.Par.OutFlagFaultDev := FALSE;
   A_3125_MXZ01MA.Mon3.Par.OutDelayTime := 0;
   A_3125_MXZ01MA.A_3125_BSA07.StCode := 0;
   A_3125_MXZ01MA.A_3125_BSA07.InMonTrue := FALSE;
   A_3125_MXZ01MA.A_3125_BSA07.InMonFalse := FALSE;
   A_3125_MXZ01MA.A_3125_BSA07.InPreAlarmTrue := FALSE;
   A_3125_MXZ01MA.A_3125_BSA07.InPreAlarmFalse := FALSE;
   A_3125_MXZ01MA.A_3125_BSA07.InStopTrueTime := FALSE;
   A_3125_MXZ01MA.A_3125_BSA07.InStopFalseTime := FALSE;
   A_3125_MXZ01MA.A_3125_BSA07.InpTrue := FALSE;
   A_3125_MXZ01MA.A_3125_BSA07.InpFaultDev := FALSE;
   A_3125_MXZ01MA.A_3125_BSA07.CmdRstTrueTime := FALSE;
   A_3125_MXZ01MA.A_3125_BSA07.CmdRstFalseTime := FALSE;
   A_3125_MXZ01MA.A_3125_BSA07.CmdRunTimeoutTime := FALSE;
   A_3125_MXZ01MA.A_3125_BSA07.CmdFaultReset := FALSE;
   A_3125_MXZ01MA.A_3125_BSA07.InLocal := FALSE;
   A_3125_MXZ01MA.A_3125_BSA07.spare0305 := FALSE;
   A_3125_MXZ01MA.A_3125_BSA07.InReport := FALSE;
   A_3125_MXZ01MA.A_3125_BSA07.OutTimeoutTime := FALSE;
   A_3125_MXZ01MA.A_3125_BSA07.InHWStop := FALSE;
   A_3125_MXZ01MA.A_3125_BSA07.InDPFault := FALSE;
   A_3125_MXZ01MA.A_3125_BSA07.OutPreAlarmTrue := FALSE;
   A_3125_MXZ01MA.A_3125_BSA07.OutPreAlarmFalse := FALSE;
   A_3125_MXZ01MA.A_3125_BSA07.OutFlagPos := FALSE;
   A_3125_MXZ01MA.A_3125_BSA07.OutFlagNeg := FALSE;
   A_3125_MXZ01MA.A_3125_BSA07.OutpFaultReset := FALSE;
   A_3125_MXZ01MA.A_3125_BSA07.OutTrue := FALSE;
   A_3125_MXZ01MA.A_3125_BSA07.StFalse := FALSE;
   A_3125_MXZ01MA.A_3125_BSA07.StCtoTrue := FALSE;
   A_3125_MXZ01MA.A_3125_BSA07.StTrue := FALSE;
   A_3125_MXZ01MA.A_3125_BSA07.StCtoFalse := FALSE;
   A_3125_MXZ01MA.A_3125_BSA07.StFault := FALSE;
   A_3125_MXZ01MA.A_3125_BSA07.OutAlarmNrLog := 0;
   A_3125_MXZ01MA.A_3125_BSA07.Par.ParObjectNo := 27130;
   A_3125_MXZ01MA.A_3125_BSA07.Par.ParMsgType := 7135;
   A_3125_MXZ01MA.A_3125_BSA07.Par.ParHornCode := 0;
   A_3125_MXZ01MA.A_3125_BSA07.Par.ParLogOff := FALSE;
   A_3125_MXZ01MA.A_3125_BSA07.Par.spare0401 := FALSE;
   A_3125_MXZ01MA.A_3125_BSA07.Par.Par2WorkingCond := TRUE;
   A_3125_MXZ01MA.A_3125_BSA07.Par.ParFaultRetry := FALSE;
   A_3125_MXZ01MA.A_3125_BSA07.Par.ParBinLevel := FALSE;
   A_3125_MXZ01MA.A_3125_BSA07.Par.ParDelayChange := 0;
   A_3125_MXZ01MA.A_3125_BSA07.Par.ParDelayTrue := 200;
   A_3125_MXZ01MA.A_3125_BSA07.Par.ParDelayFalse := 0;
   A_3125_MXZ01MA.A_3125_BSA07.Par.ParTimeoutTrue := 50;
   A_3125_MXZ01MA.A_3125_BSA07.Par.ParTimeoutFalse := 0;
   A_3125_MXZ01MA.A_3125_BSA07.Par.OutMonTime := 0;
   A_3125_MXZ01MA.A_3125_BSA07.Par.OutTransitionTime := 0;
   A_3125_MXZ01MA.A_3125_BSA07.Par.OutMonTrue := FALSE;
   A_3125_MXZ01MA.A_3125_BSA07.Par.OutMonFalse := FALSE;
   A_3125_MXZ01MA.A_3125_BSA07.Par.OutFlagFaultDev := FALSE;
   A_3125_MXZ01MA.A_3125_BSA07.Par.OutDelayTime := 0;
   A_3125_MXZ01MA.Mon5.StCode := 0;
   A_3125_MXZ01MA.Mon5.InMonTrue := FALSE;
   A_3125_MXZ01MA.Mon5.InMonFalse := FALSE;
   A_3125_MXZ01MA.Mon5.InPreAlarmTrue := FALSE;
   A_3125_MXZ01MA.Mon5.InPreAlarmFalse := FALSE;
   A_3125_MXZ01MA.Mon5.InStopTrueTime := FALSE;
   A_3125_MXZ01MA.Mon5.InStopFalseTime := FALSE;
   A_3125_MXZ01MA.Mon5.InpTrue := FALSE;
   A_3125_MXZ01MA.Mon5.InpFaultDev := FALSE;
   A_3125_MXZ01MA.Mon5.CmdRstTrueTime := FALSE;
   A_3125_MXZ01MA.Mon5.CmdRstFalseTime := FALSE;
   A_3125_MXZ01MA.Mon5.CmdRunTimeoutTime := FALSE;
   A_3125_MXZ01MA.Mon5.CmdFaultReset := FALSE;
   A_3125_MXZ01MA.Mon5.InLocal := FALSE;
   A_3125_MXZ01MA.Mon5.spare0305 := FALSE;
   A_3125_MXZ01MA.Mon5.InReport := FALSE;
   A_3125_MXZ01MA.Mon5.OutTimeoutTime := FALSE;
   A_3125_MXZ01MA.Mon5.InHWStop := FALSE;
   A_3125_MXZ01MA.Mon5.InDPFault := FALSE;
   A_3125_MXZ01MA.Mon5.OutPreAlarmTrue := FALSE;
   A_3125_MXZ01MA.Mon5.OutPreAlarmFalse := FALSE;
   A_3125_MXZ01MA.Mon5.OutFlagPos := FALSE;
   A_3125_MXZ01MA.Mon5.OutFlagNeg := FALSE;
   A_3125_MXZ01MA.Mon5.OutpFaultReset := FALSE;
   A_3125_MXZ01MA.Mon5.OutTrue := FALSE;
   A_3125_MXZ01MA.Mon5.StFalse := FALSE;
   A_3125_MXZ01MA.Mon5.StCtoTrue := FALSE;
   A_3125_MXZ01MA.Mon5.StTrue := FALSE;
   A_3125_MXZ01MA.Mon5.StCtoFalse := FALSE;
   A_3125_MXZ01MA.Mon5.StFault := FALSE;
   A_3125_MXZ01MA.Mon5.OutAlarmNrLog := 0;
   A_3125_MXZ01MA.Mon5.Par.ParObjectNo := 0;
   A_3125_MXZ01MA.Mon5.Par.ParMsgType := 0;
   A_3125_MXZ01MA.Mon5.Par.ParHornCode := 0;
   A_3125_MXZ01MA.Mon5.Par.ParLogOff := FALSE;
   A_3125_MXZ01MA.Mon5.Par.spare0401 := FALSE;
   A_3125_MXZ01MA.Mon5.Par.Par2WorkingCond := FALSE;
   A_3125_MXZ01MA.Mon5.Par.ParFaultRetry := FALSE;
   A_3125_MXZ01MA.Mon5.Par.ParBinLevel := FALSE;
   A_3125_MXZ01MA.Mon5.Par.ParDelayChange := 0;
   A_3125_MXZ01MA.Mon5.Par.ParDelayTrue := 0;
   A_3125_MXZ01MA.Mon5.Par.ParDelayFalse := 0;
   A_3125_MXZ01MA.Mon5.Par.ParTimeoutTrue := 0;
   A_3125_MXZ01MA.Mon5.Par.ParTimeoutFalse := 0;
   A_3125_MXZ01MA.Mon5.Par.OutMonTime := 0;
   A_3125_MXZ01MA.Mon5.Par.OutTransitionTime := 0;
   A_3125_MXZ01MA.Mon5.Par.OutMonTrue := FALSE;
   A_3125_MXZ01MA.Mon5.Par.OutMonFalse := FALSE;
   A_3125_MXZ01MA.Mon5.Par.OutFlagFaultDev := FALSE;
   A_3125_MXZ01MA.Mon5.Par.OutDelayTime := 0;
   A_3125_MXZ01MA.Mon6.StCode := 0;
   A_3125_MXZ01MA.Mon6.InMonTrue := FALSE;
   A_3125_MXZ01MA.Mon6.InMonFalse := FALSE;
   A_3125_MXZ01MA.Mon6.InPreAlarmTrue := FALSE;
   A_3125_MXZ01MA.Mon6.InPreAlarmFalse := FALSE;
   A_3125_MXZ01MA.Mon6.InStopTrueTime := FALSE;
   A_3125_MXZ01MA.Mon6.InStopFalseTime := FALSE;
   A_3125_MXZ01MA.Mon6.InpTrue := FALSE;
   A_3125_MXZ01MA.Mon6.InpFaultDev := FALSE;
   A_3125_MXZ01MA.Mon6.CmdRstTrueTime := FALSE;
   A_3125_MXZ01MA.Mon6.CmdRstFalseTime := FALSE;
   A_3125_MXZ01MA.Mon6.CmdRunTimeoutTime := FALSE;
   A_3125_MXZ01MA.Mon6.CmdFaultReset := FALSE;
   A_3125_MXZ01MA.Mon6.InLocal := FALSE;
   A_3125_MXZ01MA.Mon6.spare0305 := FALSE;
   A_3125_MXZ01MA.Mon6.InReport := FALSE;
   A_3125_MXZ01MA.Mon6.OutTimeoutTime := FALSE;
   A_3125_MXZ01MA.Mon6.InHWStop := FALSE;
   A_3125_MXZ01MA.Mon6.InDPFault := FALSE;
   A_3125_MXZ01MA.Mon6.OutPreAlarmTrue := FALSE;
   A_3125_MXZ01MA.Mon6.OutPreAlarmFalse := FALSE;
   A_3125_MXZ01MA.Mon6.OutFlagPos := FALSE;
   A_3125_MXZ01MA.Mon6.OutFlagNeg := FALSE;
   A_3125_MXZ01MA.Mon6.OutpFaultReset := FALSE;
   A_3125_MXZ01MA.Mon6.OutTrue := FALSE;
   A_3125_MXZ01MA.Mon6.StFalse := FALSE;
   A_3125_MXZ01MA.Mon6.StCtoTrue := FALSE;
   A_3125_MXZ01MA.Mon6.StTrue := FALSE;
   A_3125_MXZ01MA.Mon6.StCtoFalse := FALSE;
   A_3125_MXZ01MA.Mon6.StFault := FALSE;
   A_3125_MXZ01MA.Mon6.OutAlarmNrLog := 0;
   A_3125_MXZ01MA.Mon6.Par.ParObjectNo := 0;
   A_3125_MXZ01MA.Mon6.Par.ParMsgType := 0;
   A_3125_MXZ01MA.Mon6.Par.ParHornCode := 0;
   A_3125_MXZ01MA.Mon6.Par.ParLogOff := FALSE;
   A_3125_MXZ01MA.Mon6.Par.spare0401 := FALSE;
   A_3125_MXZ01MA.Mon6.Par.Par2WorkingCond := FALSE;
   A_3125_MXZ01MA.Mon6.Par.ParFaultRetry := FALSE;
   A_3125_MXZ01MA.Mon6.Par.ParBinLevel := FALSE;
   A_3125_MXZ01MA.Mon6.Par.ParDelayChange := 0;
   A_3125_MXZ01MA.Mon6.Par.ParDelayTrue := 0;
   A_3125_MXZ01MA.Mon6.Par.ParDelayFalse := 0;
   A_3125_MXZ01MA.Mon6.Par.ParTimeoutTrue := 0;
   A_3125_MXZ01MA.Mon6.Par.ParTimeoutFalse := 0;
   A_3125_MXZ01MA.Mon6.Par.OutMonTime := 0;
   A_3125_MXZ01MA.Mon6.Par.OutTransitionTime := 0;
   A_3125_MXZ01MA.Mon6.Par.OutMonTrue := FALSE;
   A_3125_MXZ01MA.Mon6.Par.OutMonFalse := FALSE;
   A_3125_MXZ01MA.Mon6.Par.OutFlagFaultDev := FALSE;
   A_3125_MXZ01MA.Mon6.Par.OutDelayTime := 0;
   A_3125_MXZ01MA.A_3125_MXZ01.StCode := 0;
   A_3125_MXZ01MA.A_3125_MXZ01.InEnableRev := FALSE;
   A_3125_MXZ01MA.A_3125_MXZ01.InEnableFwd := FALSE;
   A_3125_MXZ01MA.A_3125_MXZ01.InSlow := FALSE;
   A_3125_MXZ01MA.A_3125_MXZ01.InpRunSlow := FALSE;
   A_3125_MXZ01MA.A_3125_MXZ01.InpRunFast := FALSE;
   A_3125_MXZ01MA.A_3125_MXZ01.InpRunRev := FALSE;
   A_3125_MXZ01MA.A_3125_MXZ01.InpRunFwd := FALSE;
   A_3125_MXZ01MA.A_3125_MXZ01.InpFaultDev := FALSE;
   A_3125_MXZ01MA.A_3125_MXZ01.CmdOff := FALSE;
   A_3125_MXZ01MA.A_3125_MXZ01.CmdOn := FALSE;
   A_3125_MXZ01MA.A_3125_MXZ01.CmdNext := FALSE;
   A_3125_MXZ01MA.A_3125_MXZ01.CmdFaultReset := FALSE;
   A_3125_MXZ01MA.A_3125_MXZ01.InLocal := FALSE;
   A_3125_MXZ01MA.A_3125_MXZ01.InManual := FALSE;
   A_3125_MXZ01MA.A_3125_MXZ01.InReport := FALSE;
   A_3125_MXZ01MA.A_3125_MXZ01.InSeqStop := FALSE;
   A_3125_MXZ01MA.A_3125_MXZ01.InHWStop := FALSE;
   A_3125_MXZ01MA.A_3125_MXZ01.InDPFault := FALSE;
   A_3125_MXZ01MA.A_3125_MXZ01.OutIdling := FALSE;
   A_3125_MXZ01MA.A_3125_MXZ01.OutpRunSlow := FALSE;
   A_3125_MXZ01MA.A_3125_MXZ01.OutpRunFast := FALSE;
   A_3125_MXZ01MA.A_3125_MXZ01.OutpRunRev := FALSE;
   A_3125_MXZ01MA.A_3125_MXZ01.OutpRunFwd := FALSE;
   A_3125_MXZ01MA.A_3125_MXZ01.OutpFaultReset := FALSE;
   A_3125_MXZ01MA.A_3125_MXZ01.StStopped := FALSE;
   A_3125_MXZ01MA.A_3125_MXZ01.StStarting := FALSE;
   A_3125_MXZ01MA.A_3125_MXZ01.StStartedFwd := FALSE;
   A_3125_MXZ01MA.A_3125_MXZ01.StStopping := FALSE;
   A_3125_MXZ01MA.A_3125_MXZ01.StFault := FALSE;
   A_3125_MXZ01MA.A_3125_MXZ01.StStartedRev := FALSE;
   A_3125_MXZ01MA.A_3125_MXZ01.InOutManSlow := FALSE;
   A_3125_MXZ01MA.A_3125_MXZ01.InOutManRev := FALSE;
   A_3125_MXZ01MA.A_3125_MXZ01.OutAlarmNrLog := 0;
   A_3125_MXZ01MA.A_3125_MXZ01.Par.ParObjectNo := 27109;
   A_3125_MXZ01MA.A_3125_MXZ01.Par.ParMsgType := 7053;
   A_3125_MXZ01MA.A_3125_MXZ01.Par.ParHornCode := 10;
   A_3125_MXZ01MA.A_3125_MXZ01.Par.ParLogOff := FALSE;
   A_3125_MXZ01MA.A_3125_MXZ01.Par.ParManual := TRUE;
   A_3125_MXZ01MA.A_3125_MXZ01.Par.ParRestartDelay := FALSE;
   A_3125_MXZ01MA.A_3125_MXZ01.Par.Par2Speed := FALSE;
   A_3125_MXZ01MA.A_3125_MXZ01.Par.ParHeavyStartup := FALSE;
   A_3125_MXZ01MA.A_3125_MXZ01.Par.spare45 := FALSE;
   A_3125_MXZ01MA.A_3125_MXZ01.Par.spare46 := FALSE;
   A_3125_MXZ01MA.A_3125_MXZ01.Par.OutEdgeFaultReset := FALSE;
   A_3125_MXZ01MA.A_3125_MXZ01.Par.OutDelayFault := FALSE;
   A_3125_MXZ01MA.A_3125_MXZ01.Par.OutFlagFaultDev := FALSE;
   A_3125_MXZ01MA.A_3125_MXZ01.Par.ParMonTime := 20;
   A_3125_MXZ01MA.A_3125_MXZ01.Par.ParStartingTime := 1800;
   A_3125_MXZ01MA.A_3125_MXZ01.Par.ParStoppingTime := 1200;
   A_3125_MXZ01MA.A_3125_MXZ01.Par.ParIdlingTime := 0;
   A_3125_MXZ01MA.A_3125_MXZ01.Par.ParDelayTime := 10;
   A_3125_MXZ01MA.A_3125_MXZ01.Par.OutMonTime := 0;
   A_3125_MXZ01MA.A_3125_MXZ01.Par.OutTransitionTime := 0;
   A_3125_MXZ01MA.A_3125_MXZ01.Par.OutDelayTime := 0;
   A_3125_MXZ01MA.A_3125_MXZ01.Par.InOutManPulseLen := 0;
    A_3125_TSC01_AC.StCode := 0;
   A_3125_TSC01_AC.InMonLL := FALSE;
   A_3125_TSC01_AC.InMonL := FALSE;
   A_3125_TSC01_AC.InMonMid := FALSE;
   A_3125_TSC01_AC.InMonH := FALSE;
   A_3125_TSC01_AC.InMonHH := FALSE;
   A_3125_TSC01_AC.spare0205 := FALSE;
   A_3125_TSC01_AC.InpFaultAI := FALSE;
   A_3125_TSC01_AC.InpFaultDev := FALSE;
   A_3125_TSC01_AC.InHWStop := FALSE;
   A_3125_TSC01_AC.InDPFault := FALSE;
   A_3125_TSC01_AC.InDisable := FALSE;
   A_3125_TSC01_AC.CmdFaultReset := FALSE;
   A_3125_TSC01_AC.InLocal := FALSE;
   A_3125_TSC01_AC.spare0305 := FALSE;
   A_3125_TSC01_AC.InReport := FALSE;
   A_3125_TSC01_AC.spare0307 := FALSE;
   A_3125_TSC01_AC.OutLL := FALSE;
   A_3125_TSC01_AC.OutL := FALSE;
   A_3125_TSC01_AC.OutH := FALSE;
   A_3125_TSC01_AC.OutHH := FALSE;
   A_3125_TSC01_AC.OutOverflow := FALSE;
   A_3125_TSC01_AC.spare0405 := FALSE;
   A_3125_TSC01_AC.OutFaultAI := FALSE;
   A_3125_TSC01_AC.spare0407 := FALSE;
   A_3125_TSC01_AC.StLL := FALSE;
   A_3125_TSC01_AC.StL := FALSE;
   A_3125_TSC01_AC.StMid := FALSE;
   A_3125_TSC01_AC.StH := FALSE;
   A_3125_TSC01_AC.StHH := FALSE;
   A_3125_TSC01_AC.StFaultAI := FALSE;
   A_3125_TSC01_AC.OutWarning := FALSE;
   A_3125_TSC01_AC.OutFaulted := FALSE;
   A_3125_TSC01_AC.InpValue := 0;
   A_3125_TSC01_AC.OutValuePc := 0;
   A_3125_TSC01_AC.OutValueUnits := L#0;
   A_3125_TSC01_AC.Msg.WarningDoneLL := FALSE;
   A_3125_TSC01_AC.Msg.WarningDoneL := FALSE;
   A_3125_TSC01_AC.Msg.WarningDoneMid := FALSE;
   A_3125_TSC01_AC.Msg.WarningDoneH := FALSE;
   A_3125_TSC01_AC.Msg.WarningDoneHH := FALSE;
   A_3125_TSC01_AC.Msg.FaultDoneLL := FALSE;
   A_3125_TSC01_AC.Msg.FaultDoneL := FALSE;
   A_3125_TSC01_AC.Msg.FaultDoneMid := FALSE;
   A_3125_TSC01_AC.Msg.FaultDoneH := FALSE;
   A_3125_TSC01_AC.Msg.FaultDoneHH := FALSE;
   A_3125_TSC01_AC.Msg.FaultDoneDev := FALSE;
   A_3125_TSC01_AC.Msg.FaultDoneAI := FALSE;
   A_3125_TSC01_AC.OutAlarmNrLog := 0;
   A_3125_TSC01_AC.Par.ParObjectNo := 27111;
   A_3125_TSC01_AC.Par.ParMsgType := 7252;
   A_3125_TSC01_AC.Par.ParHornCode := 10;
   A_3125_TSC01_AC.Par.ParLogOff := FALSE;
   A_3125_TSC01_AC.Par.ParSpare0401 := FALSE;
   A_3125_TSC01_AC.Par.ParValueByUser := FALSE;
   A_3125_TSC01_AC.Par.ParLimitsPc := TRUE;
   A_3125_TSC01_AC.Par.ParWago := FALSE;
   A_3125_TSC01_AC.Par.ParNoHornByWarning := FALSE;
   A_3125_TSC01_AC.Par.ParWarningLL := FALSE;
   A_3125_TSC01_AC.Par.ParWarningL := FALSE;
   A_3125_TSC01_AC.Par.ParWarningMid := FALSE;
   A_3125_TSC01_AC.Par.ParWarningH := FALSE;
   A_3125_TSC01_AC.Par.ParWarningHH := FALSE;
   A_3125_TSC01_AC.Par.ParPreAlarmLL := FALSE;
   A_3125_TSC01_AC.Par.ParPreAlarmL := FALSE;
   A_3125_TSC01_AC.Par.ParPreAlarmMid := FALSE;
   A_3125_TSC01_AC.Par.ParPreAlarmH := FALSE;
   A_3125_TSC01_AC.Par.ParPreAlarmHH := FALSE;
   A_3125_TSC01_AC.Par.ParUnitsByZeroDigit := L#0;
   A_3125_TSC01_AC.Par.ParUnitsByMaxDigit := L#25384;
   A_3125_TSC01_AC.Par.ParUnitsBy100Pc := L#10000;
   A_3125_TSC01_AC.Par.ParLimitLL := L#-1;
   A_3125_TSC01_AC.Par.ParLimitL := L#0;
   A_3125_TSC01_AC.Par.ParLimitH := L#5400;
   A_3125_TSC01_AC.Par.ParLimitHH := L#6000;
   A_3125_TSC01_AC.Par.ParMonTimeLL := 0;
   A_3125_TSC01_AC.Par.ParMonTimeL := 0;
   A_3125_TSC01_AC.Par.ParMonTimeMid := 0;
   A_3125_TSC01_AC.Par.ParMonTimeH := 0;
   A_3125_TSC01_AC.Par.ParMonTimeHH := 0;
   A_3125_TSC01_AC.Par.ParDelayTimeDown := 10;
   A_3125_TSC01_AC.Par.ParDelayTimeUp := 10;
   A_3125_TSC01_AC.Par.ParDelayTime := 30;
   A_3125_TSC01_AC.Par.OutMonTimeLL := 0;
   A_3125_TSC01_AC.Par.OutMonTimeL := 0;
   A_3125_TSC01_AC.Par.OutMonTimeMid := 0;
   A_3125_TSC01_AC.Par.OutMonTimeH := 0;
   A_3125_TSC01_AC.Par.OutMonTimeHH := 0;
   A_3125_TSC01_AC.Par.OutDelayTimeDown := 0;
   A_3125_TSC01_AC.Par.OutDelayTimeUp := 0;
   A_3125_TSC01_AC.Par.OutDelayTime := 0;
   A_3125_TSC01_AC.Par.Spare66 := 0;
   A_3125_TSC01_AF.StCode := 0;
   A_3125_TSC01_AF.InMonLL := FALSE;
   A_3125_TSC01_AF.InMonL := FALSE;
   A_3125_TSC01_AF.InMonMid := FALSE;
   A_3125_TSC01_AF.InMonH := FALSE;
   A_3125_TSC01_AF.InMonHH := FALSE;
   A_3125_TSC01_AF.spare0205 := FALSE;
   A_3125_TSC01_AF.InpFaultAI := FALSE;
   A_3125_TSC01_AF.InpFaultDev := FALSE;
   A_3125_TSC01_AF.InHWStop := FALSE;
   A_3125_TSC01_AF.InDPFault := FALSE;
   A_3125_TSC01_AF.InDisable := FALSE;
   A_3125_TSC01_AF.CmdFaultReset := FALSE;
   A_3125_TSC01_AF.InLocal := FALSE;
   A_3125_TSC01_AF.spare0305 := FALSE;
   A_3125_TSC01_AF.InReport := FALSE;
   A_3125_TSC01_AF.spare0307 := FALSE;
   A_3125_TSC01_AF.OutLL := FALSE;
   A_3125_TSC01_AF.OutL := FALSE;
   A_3125_TSC01_AF.OutH := FALSE;
   A_3125_TSC01_AF.OutHH := FALSE;
   A_3125_TSC01_AF.OutOverflow := FALSE;
   A_3125_TSC01_AF.spare0405 := FALSE;
   A_3125_TSC01_AF.OutFaultAI := FALSE;
   A_3125_TSC01_AF.spare0407 := FALSE;
   A_3125_TSC01_AF.StLL := FALSE;
   A_3125_TSC01_AF.StL := FALSE;
   A_3125_TSC01_AF.StMid := FALSE;
   A_3125_TSC01_AF.StH := FALSE;
   A_3125_TSC01_AF.StHH := FALSE;
   A_3125_TSC01_AF.StFaultAI := FALSE;
   A_3125_TSC01_AF.OutWarning := FALSE;
   A_3125_TSC01_AF.OutFaulted := FALSE;
   A_3125_TSC01_AF.InpValue := 0;
   A_3125_TSC01_AF.OutValuePc := 0;
   A_3125_TSC01_AF.OutValueUnits := L#0;
   A_3125_TSC01_AF.Msg.WarningDoneLL := FALSE;
   A_3125_TSC01_AF.Msg.WarningDoneL := FALSE;
   A_3125_TSC01_AF.Msg.WarningDoneMid := FALSE;
   A_3125_TSC01_AF.Msg.WarningDoneH := FALSE;
   A_3125_TSC01_AF.Msg.WarningDoneHH := FALSE;
   A_3125_TSC01_AF.Msg.FaultDoneLL := FALSE;
   A_3125_TSC01_AF.Msg.FaultDoneL := FALSE;
   A_3125_TSC01_AF.Msg.FaultDoneMid := FALSE;
   A_3125_TSC01_AF.Msg.FaultDoneH := FALSE;
   A_3125_TSC01_AF.Msg.FaultDoneHH := FALSE;
   A_3125_TSC01_AF.Msg.FaultDoneDev := FALSE;
   A_3125_TSC01_AF.Msg.FaultDoneAI := FALSE;
   A_3125_TSC01_AF.OutAlarmNrLog := 0;
   A_3125_TSC01_AF.Par.ParObjectNo := 27112;
   A_3125_TSC01_AF.Par.ParMsgType := 7252;
   A_3125_TSC01_AF.Par.ParHornCode := 10;
   A_3125_TSC01_AF.Par.ParLogOff := FALSE;
   A_3125_TSC01_AF.Par.ParSpare0401 := FALSE;
   A_3125_TSC01_AF.Par.ParValueByUser := FALSE;
   A_3125_TSC01_AF.Par.ParLimitsPc := TRUE;
   A_3125_TSC01_AF.Par.ParWago := FALSE;
   A_3125_TSC01_AF.Par.ParNoHornByWarning := FALSE;
   A_3125_TSC01_AF.Par.ParWarningLL := FALSE;
   A_3125_TSC01_AF.Par.ParWarningL := FALSE;
   A_3125_TSC01_AF.Par.ParWarningMid := FALSE;
   A_3125_TSC01_AF.Par.ParWarningH := FALSE;
   A_3125_TSC01_AF.Par.ParWarningHH := FALSE;
   A_3125_TSC01_AF.Par.ParPreAlarmLL := FALSE;
   A_3125_TSC01_AF.Par.ParPreAlarmL := FALSE;
   A_3125_TSC01_AF.Par.ParPreAlarmMid := FALSE;
   A_3125_TSC01_AF.Par.ParPreAlarmH := FALSE;
   A_3125_TSC01_AF.Par.ParPreAlarmHH := FALSE;
   A_3125_TSC01_AF.Par.ParUnitsByZeroDigit := L#0;
   A_3125_TSC01_AF.Par.ParUnitsByMaxDigit := L#16880;
   A_3125_TSC01_AF.Par.ParUnitsBy100Pc := L#10000;
   A_3125_TSC01_AF.Par.ParLimitLL := L#-1;
   A_3125_TSC01_AF.Par.ParLimitL := L#3000;
   A_3125_TSC01_AF.Par.ParLimitH := L#10000;
   A_3125_TSC01_AF.Par.ParLimitHH := L#10100;
   A_3125_TSC01_AF.Par.ParMonTimeLL := 0;
   A_3125_TSC01_AF.Par.ParMonTimeL := 0;
   A_3125_TSC01_AF.Par.ParMonTimeMid := 0;
   A_3125_TSC01_AF.Par.ParMonTimeH := 0;
   A_3125_TSC01_AF.Par.ParMonTimeHH := 0;
   A_3125_TSC01_AF.Par.ParDelayTimeDown := 10;
   A_3125_TSC01_AF.Par.ParDelayTimeUp := 10;
   A_3125_TSC01_AF.Par.ParDelayTime := 30;
   A_3125_TSC01_AF.Par.OutMonTimeLL := 0;
   A_3125_TSC01_AF.Par.OutMonTimeL := 0;
   A_3125_TSC01_AF.Par.OutMonTimeMid := 0;
   A_3125_TSC01_AF.Par.OutMonTimeH := 0;
   A_3125_TSC01_AF.Par.OutMonTimeHH := 0;
   A_3125_TSC01_AF.Par.OutDelayTimeDown := 0;
   A_3125_TSC01_AF.Par.OutDelayTimeUp := 0;
   A_3125_TSC01_AF.Par.OutDelayTime := 0;
   A_3125_TSC01_AF.Par.Spare66 := 0;
   A_3125_TSC01_AT.StCode := 0;
   A_3125_TSC01_AT.InMonLL := FALSE;
   A_3125_TSC01_AT.InMonL := FALSE;
   A_3125_TSC01_AT.InMonMid := FALSE;
   A_3125_TSC01_AT.InMonH := FALSE;
   A_3125_TSC01_AT.InMonHH := FALSE;
   A_3125_TSC01_AT.spare0205 := FALSE;
   A_3125_TSC01_AT.InpFaultAI := FALSE;
   A_3125_TSC01_AT.InpFaultDev := FALSE;
   A_3125_TSC01_AT.InHWStop := FALSE;
   A_3125_TSC01_AT.InDPFault := FALSE;
   A_3125_TSC01_AT.InDisable := FALSE;
   A_3125_TSC01_AT.CmdFaultReset := FALSE;
   A_3125_TSC01_AT.InLocal := FALSE;
   A_3125_TSC01_AT.spare0305 := FALSE;
   A_3125_TSC01_AT.InReport := FALSE;
   A_3125_TSC01_AT.spare0307 := FALSE;
   A_3125_TSC01_AT.OutLL := FALSE;
   A_3125_TSC01_AT.OutL := FALSE;
   A_3125_TSC01_AT.OutH := FALSE;
   A_3125_TSC01_AT.OutHH := FALSE;
   A_3125_TSC01_AT.OutOverflow := FALSE;
   A_3125_TSC01_AT.spare0405 := FALSE;
   A_3125_TSC01_AT.OutFaultAI := FALSE;
   A_3125_TSC01_AT.spare0407 := FALSE;
   A_3125_TSC01_AT.StLL := FALSE;
   A_3125_TSC01_AT.StL := FALSE;
   A_3125_TSC01_AT.StMid := FALSE;
   A_3125_TSC01_AT.StH := FALSE;
   A_3125_TSC01_AT.StHH := FALSE;
   A_3125_TSC01_AT.StFaultAI := FALSE;
   A_3125_TSC01_AT.OutWarning := FALSE;
   A_3125_TSC01_AT.OutFaulted := FALSE;
   A_3125_TSC01_AT.InpValue := 0;
   A_3125_TSC01_AT.OutValuePc := 0;
   A_3125_TSC01_AT.OutValueUnits := L#0;
   A_3125_TSC01_AT.Msg.WarningDoneLL := FALSE;
   A_3125_TSC01_AT.Msg.WarningDoneL := FALSE;
   A_3125_TSC01_AT.Msg.WarningDoneMid := FALSE;
   A_3125_TSC01_AT.Msg.WarningDoneH := FALSE;
   A_3125_TSC01_AT.Msg.WarningDoneHH := FALSE;
   A_3125_TSC01_AT.Msg.FaultDoneLL := FALSE;
   A_3125_TSC01_AT.Msg.FaultDoneL := FALSE;
   A_3125_TSC01_AT.Msg.FaultDoneMid := FALSE;
   A_3125_TSC01_AT.Msg.FaultDoneH := FALSE;
   A_3125_TSC01_AT.Msg.FaultDoneHH := FALSE;
   A_3125_TSC01_AT.Msg.FaultDoneDev := FALSE;
   A_3125_TSC01_AT.Msg.FaultDoneAI := FALSE;
   A_3125_TSC01_AT.OutAlarmNrLog := 0;
   A_3125_TSC01_AT.Par.ParObjectNo := 27113;
   A_3125_TSC01_AT.Par.ParMsgType := 7252;
   A_3125_TSC01_AT.Par.ParHornCode := 10;
   A_3125_TSC01_AT.Par.ParLogOff := FALSE;
   A_3125_TSC01_AT.Par.ParSpare0401 := FALSE;
   A_3125_TSC01_AT.Par.ParValueByUser := FALSE;
   A_3125_TSC01_AT.Par.ParLimitsPc := TRUE;
   A_3125_TSC01_AT.Par.ParWago := FALSE;
   A_3125_TSC01_AT.Par.ParNoHornByWarning := FALSE;
   A_3125_TSC01_AT.Par.ParWarningLL := FALSE;
   A_3125_TSC01_AT.Par.ParWarningL := FALSE;
   A_3125_TSC01_AT.Par.ParWarningMid := FALSE;
   A_3125_TSC01_AT.Par.ParWarningH := FALSE;
   A_3125_TSC01_AT.Par.ParWarningHH := FALSE;
   A_3125_TSC01_AT.Par.ParPreAlarmLL := FALSE;
   A_3125_TSC01_AT.Par.ParPreAlarmL := FALSE;
   A_3125_TSC01_AT.Par.ParPreAlarmMid := FALSE;
   A_3125_TSC01_AT.Par.ParPreAlarmH := FALSE;
   A_3125_TSC01_AT.Par.ParPreAlarmHH := FALSE;
   A_3125_TSC01_AT.Par.ParUnitsByZeroDigit := L#0;
   A_3125_TSC01_AT.Par.ParUnitsByMaxDigit := L#16384;
   A_3125_TSC01_AT.Par.ParUnitsBy100Pc := L#10000;
   A_3125_TSC01_AT.Par.ParLimitLL := L#-1;
   A_3125_TSC01_AT.Par.ParLimitL := L#0;
   A_3125_TSC01_AT.Par.ParLimitH := L#7000;
   A_3125_TSC01_AT.Par.ParLimitHH := L#8000;
   A_3125_TSC01_AT.Par.ParMonTimeLL := 0;
   A_3125_TSC01_AT.Par.ParMonTimeL := 0;
   A_3125_TSC01_AT.Par.ParMonTimeMid := 0;
   A_3125_TSC01_AT.Par.ParMonTimeH := 0;
   A_3125_TSC01_AT.Par.ParMonTimeHH := 0;
   A_3125_TSC01_AT.Par.ParDelayTimeDown := 10;
   A_3125_TSC01_AT.Par.ParDelayTimeUp := 10;
   A_3125_TSC01_AT.Par.ParDelayTime := 30;
   A_3125_TSC01_AT.Par.OutMonTimeLL := 0;
   A_3125_TSC01_AT.Par.OutMonTimeL := 0;
   A_3125_TSC01_AT.Par.OutMonTimeMid := 0;
   A_3125_TSC01_AT.Par.OutMonTimeH := 0;
   A_3125_TSC01_AT.Par.OutMonTimeHH := 0;
   A_3125_TSC01_AT.Par.OutDelayTimeDown := 0;
   A_3125_TSC01_AT.Par.OutDelayTimeUp := 0;
   A_3125_TSC01_AT.Par.OutDelayTime := 0;
   A_3125_TSC01_AT.Par.Spare66 := 0;
   A_3125_TSC01_AP.StCode := 0;
   A_3125_TSC01_AP.InMonLL := FALSE;
   A_3125_TSC01_AP.InMonL := FALSE;
   A_3125_TSC01_AP.InMonMid := FALSE;
   A_3125_TSC01_AP.InMonH := FALSE;
   A_3125_TSC01_AP.InMonHH := FALSE;
   A_3125_TSC01_AP.spare0205 := FALSE;
   A_3125_TSC01_AP.InpFaultAI := FALSE;
   A_3125_TSC01_AP.InpFaultDev := FALSE;
   A_3125_TSC01_AP.InHWStop := FALSE;
   A_3125_TSC01_AP.InDPFault := FALSE;
   A_3125_TSC01_AP.InDisable := FALSE;
   A_3125_TSC01_AP.CmdFaultReset := FALSE;
   A_3125_TSC01_AP.InLocal := FALSE;
   A_3125_TSC01_AP.spare0305 := FALSE;
   A_3125_TSC01_AP.InReport := FALSE;
   A_3125_TSC01_AP.spare0307 := FALSE;
   A_3125_TSC01_AP.OutLL := FALSE;
   A_3125_TSC01_AP.OutL := FALSE;
   A_3125_TSC01_AP.OutH := FALSE;
   A_3125_TSC01_AP.OutHH := FALSE;
   A_3125_TSC01_AP.OutOverflow := FALSE;
   A_3125_TSC01_AP.spare0405 := FALSE;
   A_3125_TSC01_AP.OutFaultAI := FALSE;
   A_3125_TSC01_AP.spare0407 := FALSE;
   A_3125_TSC01_AP.StLL := FALSE;
   A_3125_TSC01_AP.StL := FALSE;
   A_3125_TSC01_AP.StMid := FALSE;
   A_3125_TSC01_AP.StH := FALSE;
   A_3125_TSC01_AP.StHH := FALSE;
   A_3125_TSC01_AP.StFaultAI := FALSE;
   A_3125_TSC01_AP.OutWarning := FALSE;
   A_3125_TSC01_AP.OutFaulted := FALSE;
   A_3125_TSC01_AP.InpValue := 0;
   A_3125_TSC01_AP.OutValuePc := 0;
   A_3125_TSC01_AP.OutValueUnits := L#0;
   A_3125_TSC01_AP.Msg.WarningDoneLL := FALSE;
   A_3125_TSC01_AP.Msg.WarningDoneL := FALSE;
   A_3125_TSC01_AP.Msg.WarningDoneMid := FALSE;
   A_3125_TSC01_AP.Msg.WarningDoneH := FALSE;
   A_3125_TSC01_AP.Msg.WarningDoneHH := FALSE;
   A_3125_TSC01_AP.Msg.FaultDoneLL := FALSE;
   A_3125_TSC01_AP.Msg.FaultDoneL := FALSE;
   A_3125_TSC01_AP.Msg.FaultDoneMid := FALSE;
   A_3125_TSC01_AP.Msg.FaultDoneH := FALSE;
   A_3125_TSC01_AP.Msg.FaultDoneHH := FALSE;
   A_3125_TSC01_AP.Msg.FaultDoneDev := FALSE;
   A_3125_TSC01_AP.Msg.FaultDoneAI := FALSE;
   A_3125_TSC01_AP.OutAlarmNrLog := 0;
   A_3125_TSC01_AP.Par.ParObjectNo := 27114;
   A_3125_TSC01_AP.Par.ParMsgType := 7252;
   A_3125_TSC01_AP.Par.ParHornCode := 10;
   A_3125_TSC01_AP.Par.ParLogOff := FALSE;
   A_3125_TSC01_AP.Par.ParSpare0401 := FALSE;
   A_3125_TSC01_AP.Par.ParValueByUser := FALSE;
   A_3125_TSC01_AP.Par.ParLimitsPc := TRUE;
   A_3125_TSC01_AP.Par.ParWago := FALSE;
   A_3125_TSC01_AP.Par.ParNoHornByWarning := FALSE;
   A_3125_TSC01_AP.Par.ParWarningLL := FALSE;
   A_3125_TSC01_AP.Par.ParWarningL := FALSE;
   A_3125_TSC01_AP.Par.ParWarningMid := FALSE;
   A_3125_TSC01_AP.Par.ParWarningH := FALSE;
   A_3125_TSC01_AP.Par.ParWarningHH := FALSE;
   A_3125_TSC01_AP.Par.ParPreAlarmLL := FALSE;
   A_3125_TSC01_AP.Par.ParPreAlarmL := FALSE;
   A_3125_TSC01_AP.Par.ParPreAlarmMid := FALSE;
   A_3125_TSC01_AP.Par.ParPreAlarmH := FALSE;
   A_3125_TSC01_AP.Par.ParPreAlarmHH := FALSE;
   A_3125_TSC01_AP.Par.ParUnitsByZeroDigit := L#0;
   A_3125_TSC01_AP.Par.ParUnitsByMaxDigit := L#16384;
   A_3125_TSC01_AP.Par.ParUnitsBy100Pc := L#10000;
   A_3125_TSC01_AP.Par.ParLimitLL := L#-1;
   A_3125_TSC01_AP.Par.ParLimitL := L#0;
   A_3125_TSC01_AP.Par.ParLimitH := L#3150;
   A_3125_TSC01_AP.Par.ParLimitHH := L#3500;
   A_3125_TSC01_AP.Par.ParMonTimeLL := 0;
   A_3125_TSC01_AP.Par.ParMonTimeL := 0;
   A_3125_TSC01_AP.Par.ParMonTimeMid := 0;
   A_3125_TSC01_AP.Par.ParMonTimeH := 0;
   A_3125_TSC01_AP.Par.ParMonTimeHH := 0;
   A_3125_TSC01_AP.Par.ParDelayTimeDown := 10;
   A_3125_TSC01_AP.Par.ParDelayTimeUp := 10;
   A_3125_TSC01_AP.Par.ParDelayTime := 30;
   A_3125_TSC01_AP.Par.OutMonTimeLL := 0;
   A_3125_TSC01_AP.Par.OutMonTimeL := 0;
   A_3125_TSC01_AP.Par.OutMonTimeMid := 0;
   A_3125_TSC01_AP.Par.OutMonTimeH := 0;
   A_3125_TSC01_AP.Par.OutMonTimeHH := 0;
   A_3125_TSC01_AP.Par.OutDelayTimeDown := 0;
   A_3125_TSC01_AP.Par.OutDelayTimeUp := 0;
   A_3125_TSC01_AP.Par.OutDelayTime := 0;
   A_3125_TSC01_AP.Par.Spare66 := 0;
   A_3126_KCU04AI1.StCode := 0;
   A_3126_KCU04AI1.InMonLL := FALSE;
   A_3126_KCU04AI1.InMonL := FALSE;
   A_3126_KCU04AI1.InMonMid := FALSE;
   A_3126_KCU04AI1.InMonH := FALSE;
   A_3126_KCU04AI1.InMonHH := FALSE;
   A_3126_KCU04AI1.spare0205 := FALSE;
   A_3126_KCU04AI1.InpFaultAI := FALSE;
   A_3126_KCU04AI1.InpFaultDev := FALSE;
   A_3126_KCU04AI1.InHWStop := FALSE;
   A_3126_KCU04AI1.InDPFault := FALSE;
   A_3126_KCU04AI1.InDisable := FALSE;
   A_3126_KCU04AI1.CmdFaultReset := FALSE;
   A_3126_KCU04AI1.InLocal := FALSE;
   A_3126_KCU04AI1.spare0305 := FALSE;
   A_3126_KCU04AI1.InReport := FALSE;
   A_3126_KCU04AI1.spare0307 := FALSE;
   A_3126_KCU04AI1.OutLL := FALSE;
   A_3126_KCU04AI1.OutL := FALSE;
   A_3126_KCU04AI1.OutH := FALSE;
   A_3126_KCU04AI1.OutHH := FALSE;
   A_3126_KCU04AI1.OutOverflow := FALSE;
   A_3126_KCU04AI1.spare0405 := FALSE;
   A_3126_KCU04AI1.OutFaultAI := FALSE;
   A_3126_KCU04AI1.spare0407 := FALSE;
   A_3126_KCU04AI1.StLL := FALSE;
   A_3126_KCU04AI1.StL := FALSE;
   A_3126_KCU04AI1.StMid := FALSE;
   A_3126_KCU04AI1.StH := FALSE;
   A_3126_KCU04AI1.StHH := FALSE;
   A_3126_KCU04AI1.StFaultAI := FALSE;
   A_3126_KCU04AI1.OutWarning := FALSE;
   A_3126_KCU04AI1.OutFaulted := FALSE;
   A_3126_KCU04AI1.InpValue := 0;
   A_3126_KCU04AI1.OutValuePc := 0;
   A_3126_KCU04AI1.OutValueUnits := L#0;
   A_3126_KCU04AI1.Msg.WarningDoneLL := FALSE;
   A_3126_KCU04AI1.Msg.WarningDoneL := FALSE;
   A_3126_KCU04AI1.Msg.WarningDoneMid := FALSE;
   A_3126_KCU04AI1.Msg.WarningDoneH := FALSE;
   A_3126_KCU04AI1.Msg.WarningDoneHH := FALSE;
   A_3126_KCU04AI1.Msg.FaultDoneLL := FALSE;
   A_3126_KCU04AI1.Msg.FaultDoneL := FALSE;
   A_3126_KCU04AI1.Msg.FaultDoneMid := FALSE;
   A_3126_KCU04AI1.Msg.FaultDoneH := FALSE;
   A_3126_KCU04AI1.Msg.FaultDoneHH := FALSE;
   A_3126_KCU04AI1.Msg.FaultDoneDev := FALSE;
   A_3126_KCU04AI1.Msg.FaultDoneAI := FALSE;
   A_3126_KCU04AI1.OutAlarmNrLog := 0;
   A_3126_KCU04AI1.Par.ParObjectNo := 27115;
   A_3126_KCU04AI1.Par.ParMsgType := 7252;
   A_3126_KCU04AI1.Par.ParHornCode := 10;
   A_3126_KCU04AI1.Par.ParLogOff := FALSE;
   A_3126_KCU04AI1.Par.ParSpare0401 := FALSE;
   A_3126_KCU04AI1.Par.ParValueByUser := FALSE;
   A_3126_KCU04AI1.Par.ParLimitsPc := TRUE;
   A_3126_KCU04AI1.Par.ParWago := FALSE;
   A_3126_KCU04AI1.Par.ParNoHornByWarning := FALSE;
   A_3126_KCU04AI1.Par.ParWarningLL := FALSE;
   A_3126_KCU04AI1.Par.ParWarningL := FALSE;
   A_3126_KCU04AI1.Par.ParWarningMid := FALSE;
   A_3126_KCU04AI1.Par.ParWarningH := TRUE;
   A_3126_KCU04AI1.Par.ParWarningHH := FALSE;
   A_3126_KCU04AI1.Par.ParPreAlarmLL := FALSE;
   A_3126_KCU04AI1.Par.ParPreAlarmL := FALSE;
   A_3126_KCU04AI1.Par.ParPreAlarmMid := FALSE;
   A_3126_KCU04AI1.Par.ParPreAlarmH := FALSE;
   A_3126_KCU04AI1.Par.ParPreAlarmHH := FALSE;
   A_3126_KCU04AI1.Par.ParUnitsByZeroDigit := L#0;
   A_3126_KCU04AI1.Par.ParUnitsByMaxDigit := L#2000;
   A_3126_KCU04AI1.Par.ParUnitsBy100Pc := L#10000;
   A_3126_KCU04AI1.Par.ParLimitLL := L#-1;
   A_3126_KCU04AI1.Par.ParLimitL := L#0;
   A_3126_KCU04AI1.Par.ParLimitH := L#3150;
   A_3126_KCU04AI1.Par.ParLimitHH := L#3550;
   A_3126_KCU04AI1.Par.ParMonTimeLL := 0;
   A_3126_KCU04AI1.Par.ParMonTimeL := 0;
   A_3126_KCU04AI1.Par.ParMonTimeMid := 0;
   A_3126_KCU04AI1.Par.ParMonTimeH := 600;
   A_3126_KCU04AI1.Par.ParMonTimeHH := 0;
   A_3126_KCU04AI1.Par.ParDelayTimeDown := 10;
   A_3126_KCU04AI1.Par.ParDelayTimeUp := 10;
   A_3126_KCU04AI1.Par.ParDelayTime := 30;
   A_3126_KCU04AI1.Par.OutMonTimeLL := 0;
   A_3126_KCU04AI1.Par.OutMonTimeL := 0;
   A_3126_KCU04AI1.Par.OutMonTimeMid := 0;
   A_3126_KCU04AI1.Par.OutMonTimeH := 0;
   A_3126_KCU04AI1.Par.OutMonTimeHH := 0;
   A_3126_KCU04AI1.Par.OutDelayTimeDown := 0;
   A_3126_KCU04AI1.Par.OutDelayTimeUp := 0;
   A_3126_KCU04AI1.Par.OutDelayTime := 0;
   A_3126_KCU04AI1.Par.Spare66 := 0;
   A_3126_KCU04AI2.StCode := 0;
   A_3126_KCU04AI2.InMonLL := FALSE;
   A_3126_KCU04AI2.InMonL := FALSE;
   A_3126_KCU04AI2.InMonMid := FALSE;
   A_3126_KCU04AI2.InMonH := FALSE;
   A_3126_KCU04AI2.InMonHH := FALSE;
   A_3126_KCU04AI2.spare0205 := FALSE;
   A_3126_KCU04AI2.InpFaultAI := FALSE;
   A_3126_KCU04AI2.InpFaultDev := FALSE;
   A_3126_KCU04AI2.InHWStop := FALSE;
   A_3126_KCU04AI2.InDPFault := FALSE;
   A_3126_KCU04AI2.InDisable := FALSE;
   A_3126_KCU04AI2.CmdFaultReset := FALSE;
   A_3126_KCU04AI2.InLocal := FALSE;
   A_3126_KCU04AI2.spare0305 := FALSE;
   A_3126_KCU04AI2.InReport := FALSE;
   A_3126_KCU04AI2.spare0307 := FALSE;
   A_3126_KCU04AI2.OutLL := FALSE;
   A_3126_KCU04AI2.OutL := FALSE;
   A_3126_KCU04AI2.OutH := FALSE;
   A_3126_KCU04AI2.OutHH := FALSE;
   A_3126_KCU04AI2.OutOverflow := FALSE;
   A_3126_KCU04AI2.spare0405 := FALSE;
   A_3126_KCU04AI2.OutFaultAI := FALSE;
   A_3126_KCU04AI2.spare0407 := FALSE;
   A_3126_KCU04AI2.StLL := FALSE;
   A_3126_KCU04AI2.StL := FALSE;
   A_3126_KCU04AI2.StMid := FALSE;
   A_3126_KCU04AI2.StH := FALSE;
   A_3126_KCU04AI2.StHH := FALSE;
   A_3126_KCU04AI2.StFaultAI := FALSE;
   A_3126_KCU04AI2.OutWarning := FALSE;
   A_3126_KCU04AI2.OutFaulted := FALSE;
   A_3126_KCU04AI2.InpValue := 0;
   A_3126_KCU04AI2.OutValuePc := 0;
   A_3126_KCU04AI2.OutValueUnits := L#0;
   A_3126_KCU04AI2.Msg.WarningDoneLL := FALSE;
   A_3126_KCU04AI2.Msg.WarningDoneL := FALSE;
   A_3126_KCU04AI2.Msg.WarningDoneMid := FALSE;
   A_3126_KCU04AI2.Msg.WarningDoneH := FALSE;
   A_3126_KCU04AI2.Msg.WarningDoneHH := FALSE;
   A_3126_KCU04AI2.Msg.FaultDoneLL := FALSE;
   A_3126_KCU04AI2.Msg.FaultDoneL := FALSE;
   A_3126_KCU04AI2.Msg.FaultDoneMid := FALSE;
   A_3126_KCU04AI2.Msg.FaultDoneH := FALSE;
   A_3126_KCU04AI2.Msg.FaultDoneHH := FALSE;
   A_3126_KCU04AI2.Msg.FaultDoneDev := FALSE;
   A_3126_KCU04AI2.Msg.FaultDoneAI := FALSE;
   A_3126_KCU04AI2.OutAlarmNrLog := 0;
   A_3126_KCU04AI2.Par.ParObjectNo := 27116;
   A_3126_KCU04AI2.Par.ParMsgType := 7252;
   A_3126_KCU04AI2.Par.ParHornCode := 10;
   A_3126_KCU04AI2.Par.ParLogOff := FALSE;
   A_3126_KCU04AI2.Par.ParSpare0401 := FALSE;
   A_3126_KCU04AI2.Par.ParValueByUser := FALSE;
   A_3126_KCU04AI2.Par.ParLimitsPc := TRUE;
   A_3126_KCU04AI2.Par.ParWago := FALSE;
   A_3126_KCU04AI2.Par.ParNoHornByWarning := FALSE;
   A_3126_KCU04AI2.Par.ParWarningLL := FALSE;
   A_3126_KCU04AI2.Par.ParWarningL := FALSE;
   A_3126_KCU04AI2.Par.ParWarningMid := FALSE;
   A_3126_KCU04AI2.Par.ParWarningH := TRUE;
   A_3126_KCU04AI2.Par.ParWarningHH := FALSE;
   A_3126_KCU04AI2.Par.ParPreAlarmLL := FALSE;
   A_3126_KCU04AI2.Par.ParPreAlarmL := FALSE;
   A_3126_KCU04AI2.Par.ParPreAlarmMid := FALSE;
   A_3126_KCU04AI2.Par.ParPreAlarmH := FALSE;
   A_3126_KCU04AI2.Par.ParPreAlarmHH := FALSE;
   A_3126_KCU04AI2.Par.ParUnitsByZeroDigit := L#0;
   A_3126_KCU04AI2.Par.ParUnitsByMaxDigit := L#2000;
   A_3126_KCU04AI2.Par.ParUnitsBy100Pc := L#10000;
   A_3126_KCU04AI2.Par.ParLimitLL := L#-1;
   A_3126_KCU04AI2.Par.ParLimitL := L#0;
   A_3126_KCU04AI2.Par.ParLimitH := L#3150;
   A_3126_KCU04AI2.Par.ParLimitHH := L#3550;
   A_3126_KCU04AI2.Par.ParMonTimeLL := 0;
   A_3126_KCU04AI2.Par.ParMonTimeL := 0;
   A_3126_KCU04AI2.Par.ParMonTimeMid := 0;
   A_3126_KCU04AI2.Par.ParMonTimeH := 600;
   A_3126_KCU04AI2.Par.ParMonTimeHH := 0;
   A_3126_KCU04AI2.Par.ParDelayTimeDown := 10;
   A_3126_KCU04AI2.Par.ParDelayTimeUp := 10;
   A_3126_KCU04AI2.Par.ParDelayTime := 30;
   A_3126_KCU04AI2.Par.OutMonTimeLL := 0;
   A_3126_KCU04AI2.Par.OutMonTimeL := 0;
   A_3126_KCU04AI2.Par.OutMonTimeMid := 0;
   A_3126_KCU04AI2.Par.OutMonTimeH := 0;
   A_3126_KCU04AI2.Par.OutMonTimeHH := 0;
   A_3126_KCU04AI2.Par.OutDelayTimeDown := 0;
   A_3126_KCU04AI2.Par.OutDelayTimeUp := 0;
   A_3126_KCU04AI2.Par.OutDelayTime := 0;
   A_3126_KCU04AI2.Par.Spare66 := 0;
   A_3126_BTE05.StCode := 0;
   A_3126_BTE05.InMonLL := FALSE;
   A_3126_BTE05.InMonL := FALSE;
   A_3126_BTE05.InMonMid := FALSE;
   A_3126_BTE05.InMonH := FALSE;
   A_3126_BTE05.InMonHH := FALSE;
   A_3126_BTE05.spare0205 := FALSE;
   A_3126_BTE05.InpFaultAI := FALSE;
   A_3126_BTE05.InpFaultDev := FALSE;
   A_3126_BTE05.InHWStop := FALSE;
   A_3126_BTE05.InDPFault := FALSE;
   A_3126_BTE05.InDisable := FALSE;
   A_3126_BTE05.CmdFaultReset := FALSE;
   A_3126_BTE05.InLocal := FALSE;
   A_3126_BTE05.spare0305 := FALSE;
   A_3126_BTE05.InReport := FALSE;
   A_3126_BTE05.spare0307 := FALSE;
   A_3126_BTE05.OutLL := FALSE;
   A_3126_BTE05.OutL := FALSE;
   A_3126_BTE05.OutH := FALSE;
   A_3126_BTE05.OutHH := FALSE;
   A_3126_BTE05.OutOverflow := FALSE;
   A_3126_BTE05.spare0405 := FALSE;
   A_3126_BTE05.OutFaultAI := FALSE;
   A_3126_BTE05.spare0407 := FALSE;
   A_3126_BTE05.StLL := FALSE;
   A_3126_BTE05.StL := FALSE;
   A_3126_BTE05.StMid := FALSE;
   A_3126_BTE05.StH := FALSE;
   A_3126_BTE05.StHH := FALSE;
   A_3126_BTE05.StFaultAI := FALSE;
   A_3126_BTE05.OutWarning := FALSE;
   A_3126_BTE05.OutFaulted := FALSE;
   A_3126_BTE05.InpValue := 0;
   A_3126_BTE05.OutValuePc := 0;
   A_3126_BTE05.OutValueUnits := L#0;
   A_3126_BTE05.Msg.WarningDoneLL := FALSE;
   A_3126_BTE05.Msg.WarningDoneL := FALSE;
   A_3126_BTE05.Msg.WarningDoneMid := FALSE;
   A_3126_BTE05.Msg.WarningDoneH := FALSE;
   A_3126_BTE05.Msg.WarningDoneHH := FALSE;
   A_3126_BTE05.Msg.FaultDoneLL := FALSE;
   A_3126_BTE05.Msg.FaultDoneL := FALSE;
   A_3126_BTE05.Msg.FaultDoneMid := FALSE;
   A_3126_BTE05.Msg.FaultDoneH := FALSE;
   A_3126_BTE05.Msg.FaultDoneHH := FALSE;
   A_3126_BTE05.Msg.FaultDoneDev := FALSE;
   A_3126_BTE05.Msg.FaultDoneAI := FALSE;
   A_3126_BTE05.OutAlarmNrLog := 0;
   A_3126_BTE05.Par.ParObjectNo := 27117;
   A_3126_BTE05.Par.ParMsgType := 7252;
   A_3126_BTE05.Par.ParHornCode := 10;
   A_3126_BTE05.Par.ParLogOff := FALSE;
   A_3126_BTE05.Par.ParSpare0401 := FALSE;
   A_3126_BTE05.Par.ParValueByUser := FALSE;
   A_3126_BTE05.Par.ParLimitsPc := TRUE;
   A_3126_BTE05.Par.ParWago := FALSE;
   A_3126_BTE05.Par.ParNoHornByWarning := FALSE;
   A_3126_BTE05.Par.ParWarningLL := FALSE;
   A_3126_BTE05.Par.ParWarningL := FALSE;
   A_3126_BTE05.Par.ParWarningMid := FALSE;
   A_3126_BTE05.Par.ParWarningH := TRUE;
   A_3126_BTE05.Par.ParWarningHH := FALSE;
   A_3126_BTE05.Par.ParPreAlarmLL := FALSE;
   A_3126_BTE05.Par.ParPreAlarmL := FALSE;
   A_3126_BTE05.Par.ParPreAlarmMid := FALSE;
   A_3126_BTE05.Par.ParPreAlarmH := FALSE;
   A_3126_BTE05.Par.ParPreAlarmHH := FALSE;
   A_3126_BTE05.Par.ParUnitsByZeroDigit := L#0;
   A_3126_BTE05.Par.ParUnitsByMaxDigit := L#27384;
   A_3126_BTE05.Par.ParUnitsBy100Pc := L#10000;
   A_3126_BTE05.Par.ParLimitLL := L#0;
   A_3126_BTE05.Par.ParLimitL := L#2000;
   A_3126_BTE05.Par.ParLimitH := L#8000;
   A_3126_BTE05.Par.ParLimitHH := L#10000;
   A_3126_BTE05.Par.ParMonTimeLL := 0;
   A_3126_BTE05.Par.ParMonTimeL := 0;
   A_3126_BTE05.Par.ParMonTimeMid := 0;
   A_3126_BTE05.Par.ParMonTimeH := 600;
   A_3126_BTE05.Par.ParMonTimeHH := 0;
   A_3126_BTE05.Par.ParDelayTimeDown := 10;
   A_3126_BTE05.Par.ParDelayTimeUp := 10;
   A_3126_BTE05.Par.ParDelayTime := 30;
   A_3126_BTE05.Par.OutMonTimeLL := 0;
   A_3126_BTE05.Par.OutMonTimeL := 0;
   A_3126_BTE05.Par.OutMonTimeMid := 0;
   A_3126_BTE05.Par.OutMonTimeH := 0;
   A_3126_BTE05.Par.OutMonTimeHH := 0;
   A_3126_BTE05.Par.OutDelayTimeDown := 0;
   A_3126_BTE05.Par.OutDelayTimeUp := 0;
